                    _TimeoutTimer(IN:=_Step > 0);
IF _TimeoutTimer.Q THEN
	_Step := 0;
	_Error := TRUE;
	_ErrorDescription := 'timed out waiting for response.';
END_IF

_ResetRtrig(CLK:=_Reset);
IF _ResetRtrig.Q THEN
	_Reset := FALSE;
	_Step := 0;
END_IF

_Done := _Step = 0;
_Busy := NOT _Done;

CASE _Step OF
	0: // IDLE
		IF _Execute AND NOT _PythonTcpClient.bBusyWrite THEN
			_Execute := FALSE;
			_Step := _Step + 1;
		ELSIF _Execute THEN
			_Execute := FALSE;
		END_IF
	
	1: // CALL
		_ReadRecordLast := _PythonTcpClient.bRecordRead;
		IF _PythonTcpClient.M_Write(Data:=_Command) THEN
			_Step := _Step + 1;
		ELSE
			_Error := TRUE;
			_ErrorDescription := 'tcp client busy or not connected';
			_Step := 0;
		END_IF
	
	2: // WAIT
		IF _PythonTcpClient.bRecordRead <> _ReadRecordLast THEN
			_ReadRecordLast := _PythonTcpClient.bRecordRead;
			IF find(_PythonTcpClient.strRead, 'res: ') = 1 THEN
				MemUtils.MemSet(
					pbyBuffer:=ADR(_Response),
					byValue:=0,
					dwSize:=SIZEOF(_Response));
				_Response := _PythonTcpClient.strRead;
				_Step := 0;
				
			ELSIF find(_PythonTcpClient.strRead, 'worker uid: ') = 1 THEN
				MemUtils.MemSet(
					pbyBuffer:=ADR(_WorkerUid),
					byValue:=0,
					dwSize:=SIZEOF(_WorkerUid));
				_WorkerUid := DELETE(STR:=_PythonTcpClient.strRead, LEN:=12, POS:=1);
				
			ELSIF find(_PythonTcpClient.strRead, 'command uid: ') = 1 THEN
				MemUtils.MemSet(
					pbyBuffer:=ADR(_WorkerUid),
					byValue:=0,
					dwSize:=SIZEOF(_WorkerUid));
				_WorkerUid := DELETE(STR:=_PythonTcpClient.strRead, LEN:=12, POS:=1);
				
			END_IF
		END_IF
		
END_CASE

_PythonTcpClient(
	bEnable:= TRUE, 
	strIpAddress:= sIpAddress, 
	uPort:= uPort,
	bBusyWrite=> , 
	bDoneWrite=> , 
	bBusyRead=> , 
	bRecordRead=> , 
	strRead=> );
                  

METHOD PUBLIC M_Reset : BOOL
VAR_INPUT
END_VAR
                          _Reset := TRUE;
_Error := FALSE;
_ErrorDescription := '';
                        
END_METHOD

METHOD PUBLIC M_CalibrateCamera : BOOL
VAR_INPUT
	iImageWidth: UINT:=2016;
	iImageHeight: UINT:=2000;
	uTimeout: UDINT:=60; //sec
	fCalCheckerSize: REAL:=25.0; //mm
	iCalCheckerX: UINT:=6;
	iCalCheckerY: UINT:=9;
END_VAR
VAR	
	_CalScriptFileName: STRING:='/var/opt/codesys/PlcLogic/Application/Vision/CalibrateCamera.py';
	_CalResultFile: STRING:='/var/opt/codesys/PlcLogic/visu/outputimage.jpg';
END_VAR
                          
// calibrate with a checkerboard
// sudo python /var/opt/codesys/PlcLogic/Application/CalibrateCamera.py -s cal.yaml -l 24.5 -x 6 -y 9 -d false

IF NOT _Busy THEN
	M_CalibrateCamera := TRUE;
	
	_TimeoutTimer.PT := UDINT_TO_TIME(uTimeout * 1000);
	
	_Command := CONCAT('sudo python ', _CalScriptFileName);
	_Command := CONCAT(_Command, ' -l ');
	_Command := CONCAT(_Command, REAL_TO_STRING(fCalCheckerSize));
	_Command := CONCAT(_Command, ' -x ');
	_Command := CONCAT(_Command, UINT_TO_STRING(iCalCheckerX));
	_Command := CONCAT(_Command, ' -y ');
	_Command := CONCAT(_Command, UINT_TO_STRING(iCalCheckerY));
	_Command := CONCAT(_Command, ' -w ');
	_Command := CONCAT(_Command, UINT_TO_STRING(iImageWidth));
	_Command := CONCAT(_Command, ' -h ');
	_Command := CONCAT(_Command, UINT_TO_STRING(iImageHeight));
	_Command := CONCAT(_Command, ' -r ');
	_Command := CONCAT(_Command, _CalResultFile);
	_Command := CONCAT(_Command, ' 2> ./vision_log.txt ');
	_Execute := TRUE;
	
ELSE
	M_CalibrateCamera := FALSE;
	//_Error := TRUE;
	//_ErrorDescription := 'function busy.';
	
END_IF
                        
END_METHOD

METHOD PUBLIC M_Cancel : BOOL
VAR_INPUT
END_VAR
                          IF _WorkerUid <> '' THEN
	M_Cancel := TRUE;
	_Command := 'kill: ';
	_Command := CONCAT(_Command, _WorkerUid);
	_WorkerUid := ''; // lets make sure to forget this uid in case its used again for something else
	_Step := 0;
	_Execute := TRUE;
	
ELSE
	M_Cancel := FALSE;
	
END_IF
                        
END_METHOD

METHOD PUBLIC M_CaptureImage : BOOL
VAR_INPUT
	iImageWidth: UINT:=2016;
	iImageHeight: UINT:=2000;
	uTimeout: UDINT:=60; //sec
END_VAR
VAR
	_ImageScriptFileName: STRING:='/var/opt/codesys/PlcLogic/Application/Vision/CaptureImage.py';
	_CaptureImageName: STRING:='/var/opt/codesys/PlcLogic/visu/outputimage.jpg';
END_VAR
                          
// capture an image
// sudo python /var/opt/codesys/PlcLogic/Application/CaptureImage.py -s /var/opt/codesys/PlcLogic/Application/input.jpg -w 2016 -h 2000

IF NOT _Busy THEN
	M_CaptureImage := TRUE;
	
	_TimeoutTimer.PT := UDINT_TO_TIME(uTimeout * 1000);
	
	_Command := CONCAT('sudo python ', _ImageScriptFileName);
	_Command := CONCAT(_Command, ' -s ');
	_Command := CONCAT(_Command, _CaptureImageName);
	_Command := CONCAT(_Command, ' -w ');
	_Command := CONCAT(_Command, UINT_TO_STRING(iImageWidth));
	_Command := CONCAT(_Command, ' -h ');
	_Command := CONCAT(_Command, UINT_TO_STRING(iImageHeight));
	_Command := CONCAT(_Command, ' 2> ./vision_log.txt '); 
	_Execute := TRUE;
	
ELSE
	M_CaptureImage := FALSE;
	//_Error := TRUE;
	//_ErrorDescription := 'function busy.';
	
END_IF

                        
END_METHOD

METHOD PUBLIC M_LocatePart : BOOL
VAR_INPUT
	iImageWidth: UINT:=2016;
	iImageHeight: UINT:=2000;
	uTimeout: UDINT:=60; //sec
	iMaxPos: UINT:=10; // i
	dMaxOverlap: REAL:=0.0; // j
	dScore: REAL:=0.8; // k
	dToleranceAngle: REAL:=90.0; // l
	sTemplateName: STRING:='template.jpg';
	sScriptFilename: STRING:='FastTemplateMatching.py';
END_VAR
VAR CONSTANT
	//_SCRIPT_FILE_NAME: STRING:='/var/opt/codesys/PlcLogic/Application/Vision/FastTemplateMatching.py';
	_SCRIPT_DIR_PATH: STRING:='/var/opt/codesys/PlcLogic/Application/Vision/';
	_RESULT_FILE_NAME: STRING:='/var/opt/codesys/PlcLogic/visu/outputimage.jpg';
	_TEMPLATE_DIR_PATH: STRING:='/var/opt/codesys/PlcLogic/Application/Vision/Templates/';
END_VAR
                          
// run the designated vision program
// sudo python /var/opt/codesys/PlcLogic/Application/Vision/TemplateMatch.py -s /var/opt/codesys/PlcLogic/visu/outputimage.jpg        -t /var/opt/codesys/PlcLogic/Application/Vision/Template3.JPG -i 0.9 -j 1.0 -d true -w 2016 -h 2000
// sudo python /var/opt/codesys/PlcLogic/Application/Vision/FastTemplateMatching.py -s /var/opt/codesys/PlcLogic/visu/outputimage.jpg -t /var/opt/codesys/PlcLogic/Application/Vision/Template.jpg -w 2016 -h 2000 -d false
IF NOT _Busy THEN
	M_LocatePart := TRUE;
	
	_TimeoutTimer.PT := UDINT_TO_TIME(uTimeout * 1000);
	
	_Command := CONCAT('sudo python ', _SCRIPT_DIR_PATH);
	_Command := CONCAT(_Command, sScriptFilename);
	//_Command := CONCAT(_Command, ' -s '); // need to trim down the string length
	//_Command := CONCAT(_Command, _VisionImageName);
	_Command := CONCAT(_Command, ' -t ');
	_Command := CONCAT(_Command, _TEMPLATE_DIR_PATH);
	_Command := CONCAT(_Command, sTemplateName);
	_Command := CONCAT(_Command, ' -i ');
	_Command := CONCAT(_Command, UINT_TO_STRING(iMaxPos));
	_Command := CONCAT(_Command, ' -j ');
	_Command := CONCAT(_Command, REAL_TO_STRING(dMaxOverlap));
	_Command := CONCAT(_Command, ' -k ');
	_Command := CONCAT(_Command, REAL_TO_STRING(dScore));
	_Command := CONCAT(_Command, ' -l ');
	_Command := CONCAT(_Command, REAL_TO_STRING(dToleranceAngle));
	_Command := CONCAT(_Command, ' -w ');
	_Command := CONCAT(_Command, UINT_TO_STRING(iImageWidth));
	_Command := CONCAT(_Command, ' -h ');
	_Command := CONCAT(_Command, UINT_TO_STRING(iImageHeight));
	_Command := CONCAT(_Command, ' 2> ./vision_log.txt ');
	_Execute := TRUE;
	
ELSE
	M_LocatePart := FALSE;
	//_Error := TRUE;
	//_ErrorDescription := 'function busy.';
	
END_IF
                        
END_METHOD

{attribute 'monitoring':='variable'}
PROPERTY PUBLIC P_Busy : BOOL
GET
VAR
END_VAR
                            P_Busy := _Busy;
                          
END_GET
END_PROPERTY

{attribute 'monitoring':='variable'}
PROPERTY PUBLIC P_Done : BOOL
GET
VAR
END_VAR
                            P_Done := _Done;
                          
END_GET
END_PROPERTY

{attribute 'monitoring':='variable'}
PROPERTY PUBLIC P_Result : STRING(255)
GET
VAR
END_VAR
                            P_Result := _Response;
                          
END_GET
END_PROPERTY

PROPERTY PUBLIC P_Error : BOOL
GET
VAR
END_VAR
                            P_Error := _Error;
                          
END_GET
END_PROPERTY

PROPERTY PUBLIC P_ErrorDescription : STRING
GET
VAR
END_VAR
                            P_ErrorDescription := _ErrorDescription;
                          
END_GET
END_PROPERTY
END_FUNCTION_BLOCK

FUNCTION_BLOCK PythonTcpClient
VAR_INPUT
	bEnable: BOOL;
	strIpAddress: STRING(19):='127.0.0.1';
	uPort: UINT:=50011;
END_VAR
VAR
	_Write: BOOL:=FALSE;
	_DataToWrite: STRING(255):='';
END_VAR
VAR_OUTPUT
	bBusyWrite: BOOL;
	bDoneWrite: BOOL;
	bBusyRead: BOOL;
	bRecordRead: DINT;
	strRead: STRING(255);
	bConnected: BOOL;
END_VAR

VAR
    _ipAddress       : NBS.IPv4Address;
    _fbTcpClient     : NBS.TCP_Client;
    _fbTcpRead       : NBS.TCP_Read;
    _fbTcpWrite      : NBS.TCP_Write;	
	
	_ConnectDelayTimer: TON;
	_WriteRetriesMax: INT:=3;
	_WriteRetriesCount: INT;
	_WriteRetry: BOOL;
	
	_WriteData: StringByteArray;
	_ReadData: StringByteArray;
	//_TxString: STRING(255);
	//_RxString: STRING(255);
	
	_WriteRTRIG: R_TRIG;
	_ConnectStep, _WriteStep, _ReadStep: INT;
	_Read: BOOL;
END_VAR

VAR CONSTANT
	ConnectStep_IDLE: 	INT:=00;
	ConnectStep_DELAY: 	INT:=10;
	ConnectStep_SETUP: 	INT:=20;
	ConnectStep_ENABLE: INT:=30;
	ConnectStep_WAIT: 	INT:=40;
	ConnectStep_CONN: 	INT:=50;
END_VAR

VAR CONSTANT
	WriteStep_IDLE: 	INT:=00;
	WriteStep_DATA: 	INT:=10;
	WriteStep_WRITE: 	INT:=20;
	WriteStep_WAIT: 	INT:=30;
END_VAR

VAR CONSTANT
	ReadStep_RESET: 	INT:=00;
	ReadStep_IDLE: 		INT:=10;
	ReadStep_ENABLE: 	INT:=20;
	ReadStep_MONITOR: 	INT:=30;
END_VAR

                    {region "connect"}
	
	bConnected := (_ConnectStep = ConnectStep_CONN);
	_ConnectDelayTimer(IN:=_ConnectStep = ConnectStep_DELAY, PT:=T#1S);
	CASE _ConnectStep OF
		
		ConnectStep_IDLE: // IDLE
			IF bEnable THEN
				_fbTcpClient.xEnable := FALSE;
				_ConnectStep := ConnectStep_DELAY;
			END_IF
			
		ConnectStep_DELAY: // DELAY
			IF _ConnectDelayTimer.Q THEN
				_ConnectStep := ConnectStep_SETUP;
			END_IF
			
		ConnectStep_SETUP: // SETUP
			_ipAddress.SetInitialValue(ipAddress := strIpAddress);
			_ConnectStep := ConnectStep_ENABLE;
			
		ConnectStep_ENABLE: // ENABLE
			_fbTcpClient.xEnable := TRUE;
			_ConnectStep := ConnectStep_WAIT;
			
		ConnectStep_WAIT: // WAIT
			IF _fbTcpClient.xActive THEN
				_ConnectStep := ConnectStep_CONN;
			ELSIF _fbTcpClient.xError THEN
				_ConnectStep := ConnectStep_IDLE;
			END_IF
		
		ConnectStep_CONN: // CONNECTED
			IF _fbTcpClient.xError OR NOT _fbTcpClient.xActive OR NOT bEnable THEN
				_ConnectStep := ConnectStep_IDLE;
			END_IF
			
	END_CASE
	
	_fbTcpClient(
		xEnable := , 
		itfIPAddress := _ipAddress, 
		uiPort := uPort, 
		udiTimeOut := 1000000); // us
			 
{endregion}


{region "write"}
	_WriteRTRIG(CLK:=_Write);
	CASE _WriteStep OF
			
		WriteStep_IDLE: // IDLE
			IF (_WriteRTRIG.Q OR _WriteRetry) AND bConnected THEN
				_Write := FALSE;
				_WriteRetry := FALSE;
				_fbTcpWrite.xExecute := FALSE;
				_WriteStep := WriteStep_DATA;
			END_IF
			
		WriteStep_DATA: // DATA
			IF _DataToWrite <> '' THEN
				MemUtils.MemSet(
					pbyBuffer:=ADR(_WriteData.bArray),
					byValue:=0,
					dwSize:=SIZEOF(_WriteData.bArray));
				MemUtils.MemCpy(
					pbyDest:=ADR(_WriteData.sString),
					pbySrc:=ADR(_DataToWrite),
					dwSize:=INT_TO_DWORD(LEN(_DataToWrite)));
				_WriteStep := WriteStep_WRITE;
			ELSE
				_WriteStep := WriteStep_IDLE;
			END_IF
			
		WriteStep_WRITE: // WRITE
			_fbTcpWrite.xExecute := TRUE;
			_WriteStep := WriteStep_WAIT;
		
		WriteStep_WAIT: // WAIT
			IF _fbTcpWrite.xDone THEN
				_fbTcpWrite.xExecute := FALSE;
				_WriteRetriesCount := 0;
				_WriteStep := WriteStep_IDLE;
				
			ELSIF _fbTcpWrite.xError THEN
				IF _WriteRetriesCount <= _WriteRetriesMax THEN
					_WriteRetriesCount := _WriteRetriesCount + 1;
					_WriteRetry := TRUE;
					_WriteStep := WriteStep_IDLE;
					
				ELSIF _WriteRetriesCount > _WriteRetriesMax THEN
					_WriteRetriesCount := 0;
					_WriteStep := WriteStep_IDLE;
					
				END_IF
			END_IF
	END_CASE
	
	bBusyWrite := ((_WriteStep <> WriteStep_IDLE) OR _WriteRetry) AND _fbTcpWrite.xBusy;
	bDoneWrite := (_WriteStep = WriteStep_IDLE) AND _fbTcpWrite.xDone;
	_fbTcpWrite(xExecute := ,
				itfConnection := _fbTcpClient.itfConnection, 
				udiTimeOut := 1000000, // us 
				udiSize := INT_TO_UDINT(LEN(_WriteData.sString)), 
				pData := ADR(_WriteData.bArray));

{endregion}


{region "read"}

	_Read := (_ConnectStep = ConnectStep_CONN);
	CASE _ReadStep OF
			 
		ReadStep_RESET: // RESET
			_fbTcpRead.xEnable := FALSE;
			_ReadStep := ReadStep_IDLE;

		ReadStep_IDLE: // IDLE
			IF _Read THEN
				_ReadStep := ReadStep_ENABLE;
			END_IF

		ReadStep_ENABLE: // ENABLE
			_fbTcpRead.xEnable := TRUE;
			_ReadStep := ReadStep_MONITOR;

		ReadStep_MONITOR: // MONITOR
			IF _fbTcpRead.xReady THEN
				IF (_fbTcpRead.udiCount > 0) THEN
					//
					MemUtils.MemSet(
						pbyBuffer:=ADR(strRead),
						byValue:=0,
						dwSize:=SIZEOF(strRead)); 
					MemUtils.MemCpy(
						pbyDest:=ADR(strRead),
						pbySrc:=ADR(_ReadData.sString),
						dwSize:=SEL(_fbTcpRead.udiCount > 255, _fbTcpRead.udiCount, 255));
					MemUtils.MemSet(
						pbyBuffer:=ADR(_ReadData.sString),
						byValue:=0,
						dwSize:=SIZEOF(_ReadData.sString)); 
					//
					bRecordRead := bRecordRead + 1;
				END_IF
				
			ELSIF _fbTcpRead.xError OR NOT _Read THEN
				_ReadStep := ReadStep_RESET;
				
			END_IF
			 
	END_CASE
	
	bBusyRead := (_ReadStep <> ReadStep_IDLE) AND _fbTcpRead.xBusy;
	_fbTcpRead(xEnable := , 
				itfConnection := _fbTcpClient.itfConnection, 
				udiSize := SIZEOF(_ReadData.bArray), 
				pData := ADR(_ReadData.bArray), 
				udiCount => );

{endregion}
                  

METHOD PUBLIC M_Write : BOOL
VAR_INPUT
	Data: STRING(255);
END_VAR
                          IF bConnected AND NOT bBusyWrite THEN
	_Write:=TRUE;
	_DataToWrite:=Data;
	M_Write := TRUE;
	
ELSE
	M_Write := FALSE;
	
END_IF
                        
END_METHOD
END_FUNCTION_BLOCK

FUNCTION_BLOCK ParseVisionCmd
VAR_INPUT
    Command: STRING(GVL.COMMAND_LEN);
END_VAR
VAR_OUTPUT
    stCommand: ST_VisionCmd;
	Error: BOOL;
	ErrorDescription: STRING;
END_VAR
VAR
	_CmdParams: ARRAY [0..GVL.COMMAND_LEN] OF STRING;
    _CommandType: STRING;
	_StrPosition: INT;
END_VAR
VAR CONSTANT
	_CommandTypeCal: STRING(3):='CAL'; // calibrate vision
	_CommandTypeAcq: STRING(3):='ACQ'; // acquire (capture) image
	_CommandTypeLoc: STRING(3):='LOC'; // locate part
END_VAR

                    // C|A|L ImageWidth ImageHeight Timeout

// C Calibrate vision system
    // CheckerSize (user units) XCount YCount 
    // C 2016 2000 60 25.0 6 9
    
// A Aquire image
    // A 2016 2000 60
    
// L Locate part 
    // MaxParts MaxOverlap Score ToleranceAngle ResultPostion TemplateName ScriptName
    // L 2016 2000 60 10 0.0 0.8 90.0 1 template.jpg FastTemplateMatching.py
	// MaxParts - max number of parts to find in image
	// MaxOverlap - max overlap of parts in image
	// Score - min required score for parts
	// ToleranceAngle - +/- search angle (the larger the number, the longer the search)
	// ResultPostion - index of vision register to store result
	// TemplateName - name of the template to search for
	// ScriptName - name of the template to search for

Error:=FALSE;
ErrorDescription:='';

// split command string into commands
_CmdParams:=F_SplitCmd(Command:=Command);

_CommandType:= _CmdParams[0];
IF _CommandType = _CommandTypeCal THEN
    // C 2016 2000 0060 025.0 0006 0009
	stCommand.CommandType:=DUT_Command_VisionType.Calibrate;
    stCommand.Calibrate.CheckerSize:=STRING_TO_REAL(_CmdParams[4]);
    stCommand.Calibrate.CheckerXCount:=STRING_TO_UINT(_CmdParams[5]);
    stCommand.Calibrate.CheckerYCount:=STRING_TO_UINT(_CmdParams[6]);
	
	IF stCommand.Calibrate.CheckerSize <= 0
		OR stCommand.Calibrate.CheckerXCount <= 0
		OR stCommand.Calibrate.CheckerYCount <= 0 THEN
			Error:=TRUE;
			ErrorDescription:='Checkerboard configuration incorrect';
			RETURN;
	END_IF
    
ELSIF _CommandType = _CommandTypeAcq THEN
    // A 2016 2000 0060
	stCommand.CommandType:=DUT_Command_VisionType.Acquire;
    
ELSIF _CommandType = _CommandTypeLoc THEN
    // L 2016 2000 0060 0010 000.0 0.8 090.0 001 template.jpg FastTemplatMatching.py
	stCommand.CommandType:=DUT_Command_VisionType.LocatePart;
    stCommand.Locate.MaxParts:=STRING_TO_UINT(_CmdParams[4]);
    stCommand.Locate.MaxOverlap:=STRING_TO_REAL(_CmdParams[5]);
    stCommand.Locate.Score:=STRING_TO_REAL(_CmdParams[6]);
    stCommand.Locate.ToleranceAngle:=STRING_TO_REAL(_CmdParams[7]);
    stCommand.Locate.ResultPosition:=STRING_TO_UINT(_CmdParams[8]);
    stCommand.Locate.TemplateName:=_CmdParams[9];
    stCommand.Locate.ScriptFilename:=_CmdParams[10];
	
	IF stCommand.Locate.MaxParts <= 0
		OR stCommand.Locate.ResultPosition < GVL.VIS_ARR_BEG
		OR stCommand.Locate.ResultPosition > GVL.VIS_ARR_END
		OR stCommand.Locate.TemplateName = '' THEN
			Error:=TRUE;
			ErrorDescription:='Locate part configuration incorrect';
			RETURN;
	END_IF
	
ELSE
	Error:=TRUE;
	ErrorDescription:='Unknown command type for vision';
	RETURN;
    
END_IF

// common
stCommand.ImageWidth:=STRING_TO_UINT(_CmdParams[1]);
stCommand.ImageHeight:=STRING_TO_UINT(_CmdParams[2]);
stCommand.Timeout:=STRING_TO_UDINT(_CmdParams[3]);

IF stCommand.ImageWidth <= 0
	OR stCommand.ImageHeight <= 0 THEN
		Error:=TRUE;
		ErrorDescription:='Image size settings incorrect';
END_IF
                  
END_FUNCTION_BLOCK

FUNCTION BuildVisionCmd : STRING(GVL.COMMAND_LEN)
VAR_INPUT
    stCommand: ST_VisionCmd;
END_VAR
VAR
    _Command: STRING(GVL.COMMAND_LEN);
END_VAR
VAR CONSTANT
	_Delimiter: STRING:=' ';
	_CommandTypeCal: STRING(3):='CAL'; // calibrate vision
	_CommandTypeAcq: STRING(3):='ACQ'; // acquire (capture) image
	_CommandTypeLoc: STRING(3):='LOC'; // locate part
END_VAR

                    // C|A|L ImageWidth ImageHeight Timeout

// C Calibrate vision system
    // CheckerSize (user units) XCount YCount 
    // C 2016 2000 60 25.0 6 9
    
// A Aquire image
    // A 2016 2000 60
    
// L Locate part 
    // MaxParts MaxOverlap Score ToleranceAngle ResultPostion TemplateName ScriptName
    // L 2016 2000 60 10 0.0 0.8 90.0 1 template.jpg FastTemplateMatching.py
	// MaxParts - max number of parts to find in image
	// MaxOverlap - max overlap of parts in image
	// Score - min required score for parts
	// ToleranceAngle - +/- search angle (the larger the number, the longer the search)
	// ResultPostion - index of vision register to store result
	// TemplateName - name of the template to search for
	// ScriptName - name of the template to search for

// clear the command
_Command:='';

// build the command
CASE stCommand.CommandType OF
	DUT_Command_VisionType.Calibrate:
		F_AddElement(_Command, _Delimiter, _CommandTypeCal);
	DUT_Command_VisionType.Acquire:
		F_AddElement(_Command, _Delimiter, _CommandTypeAcq);
	DUT_Command_VisionType.LocatePart:
		F_AddElement(_Command, _Delimiter, _CommandTypeLoc);
END_CASE

// add the common items width, height, timeout
F_AddElement(_Command, _Delimiter, UINT_TO_STRING(stCommand.ImageWidth));
F_AddElement(_Command, _Delimiter, UINT_TO_STRING(stCommand.ImageHeight));
F_AddElement(_Command, _Delimiter, UDINT_TO_STRING(stCommand.Timeout));

//
CASE stCommand.CommandType OF
	DUT_Command_VisionType.Calibrate:
		// C 2016 2000 60 25.0 6 9
		F_AddElement(_Command, _Delimiter, REAL_TO_STRING(stCommand.Calibrate.CheckerSize));
		F_AddElement(_Command, _Delimiter, UINT_TO_STRING(stCommand.Calibrate.CheckerXCount));
		F_AddElement(_Command, _Delimiter, UINT_TO_STRING(stCommand.Calibrate.CheckerYCount));
		
	DUT_Command_VisionType.Acquire:
		// A 2016 2000 60
		// we are done
		
	DUT_Command_VisionType.LocatePart:
		// L 2016 2000 60 10 0.0 0.8 90.0 1 template.jpg FastTemplateMatching.py
		F_AddElement(_Command, _Delimiter, UINT_TO_STRING(stCommand.Locate.MaxParts));
		F_AddElement(_Command, _Delimiter, REAL_TO_STRING(stCommand.Locate.MaxOverlap));
		F_AddElement(_Command, _Delimiter, REAL_TO_STRING(stCommand.Locate.Score));
		F_AddElement(_Command, _Delimiter, REAL_TO_STRING(stCommand.Locate.ToleranceAngle));
		F_AddElement(_Command, _Delimiter, UINT_TO_STRING(stCommand.Locate.ResultPosition));
		F_AddElement(_Command, _Delimiter, stCommand.Locate.TemplateName);
		F_AddElement(_Command, _Delimiter, stCommand.Locate.ScriptFilename);
		
END_CASE

// set function equal to command
BuildVisionCmd := _Command;
                  
END_FUNCTION

FUNCTION_BLOCK Module EXTENDS PackML IMPLEMENTS ItfModule

VAR_INPUT // input vars
	StoredPositions: REFERENCE TO ARRAY[GVL.POS_ARR_BEG..GVL.POS_ARR_END] OF DUT_StoredPosition;
	VisionRegisters: REFERENCE TO ARRAY[GVL.VIS_ARR_BEG..GVL.VIS_ARR_END] OF DUT_VisionRegister;
	Flags: REFERENCE TO ARRAY[GVL.FLG_ARR_BEG..GVL.FLG_ARR_END] OF DUT_Flags;
END_VAR

VAR_OUTPUT // output vars
	ItfUnitMode: PACK_ML.IUnitMode;
	Busy: BOOL;
	Error: BOOL;
	ErrorDescription: STRING;
END_VAR

VAR // standard local vars
	_TimeoutTimer: TON:=(PT:=T#120S);
	_Home, _Start: BOOL;
	_ModuleFirstScan: BOOL:=TRUE;
	_SeqStart, _SeqHome: INT;
	_AbortedRtrig: R_Trig;
END_VAR

VAR CONSTANT //
	STEP_IDLE: INT := 0000;
	STEP_DONE: INT := 0020;
	STEP_RUN:  INT := 0030;
END_VAR

                    SUPER^();

//
IF _ModuleFirstScan THEN
	ItfUnitMode := SUPER^.IUnitMode;
END_IF;

//
_M_Home();
_M_Start();

//
Busy := _UnitMode.CurrentState <> PACK_ML.State.Idle
		AND _UnitMode.CurrentState <> PACK_ML.State.Aborted
		AND _UnitMode.CurrentState <> PACK_ML.State.Complete
		AND _UnitMode.CurrentState <> PACK_ML.State.Held
		AND _UnitMode.CurrentState <> PACK_ML.State.Stopped
		AND _UnitMode.CurrentState <> PACK_ML.State.Suspended;
		
//
_AbortedRtrig(CLK:=_UnitMode.CurrentState = PACK_ML.State.Aborted);
IF _AbortedRtrig.Q THEN
	//_SeqStart := 0;  _Start:=FALSE;
	//_SeqHome := 0; _Home:=FALSE;
END_IF

//
_TimeoutTimer(IN:= Busy);
IF _TimeoutTimer.Q THEN
	M_Error(Description:= CONCAT('Task timed out after ', TIME_TO_STRING(_TimeoutTimer.ET)));
END_IF

// do not place anything below this
_ModuleFirstScan:=FALSE;
                  

METHOD PUBLIC M_Start
VAR_INPUT
END_VAR
                          _Start := TRUE;
                        
END_METHOD

METHOD PUBLIC M_Home
VAR_INPUT
END_VAR
                          _Home:=TRUE;
                        
END_METHOD

METHOD PROTECTED M_Error : BOOL
VAR_INPUT
	Description: STRING;
END_VAR
                          // suspend state machine
_UnitMode.Suspend();

//
Error := TRUE;

//
IF ErrorDescription = '' THEN
	ErrorDescription := Description;
ELSE // add a space and tack on the additional error description
	ErrorDescription := CONCAT(ErrorDescription, ' ');
	ErrorDescription := CONCAT(ErrorDescription, Description);
END_IF
                        
END_METHOD

METHOD PUBLIC M_Abort
VAR_INPUT
END_VAR
                          _UnitMode.Abort();
_SeqStart := 0;  _Start:=FALSE;
_SeqHome := 0; _Home:=FALSE;
                        
END_METHOD

METHOD PUBLIC M_Hold
VAR_INPUT
END_VAR
                          _UnitMode.Hold();
                        
END_METHOD

METHOD PUBLIC M_Stop
VAR_INPUT
END_VAR
                          _UnitMode.Stop();
                        
END_METHOD

METHOD PRIVATE _M_Start : BOOL
                          CASE _SeqStart OF
	0:
		IF _Start THEN
			_Start := FALSE;
			M_Reset();
			_SeqStart := _SeqStart + 1;
		END_IF
	1:
		CASE _UnitMode.CurrentState OF
			PACK_ML.State.Clearing,
			PACK_ML.State.Resetting,
			PACK_ML.State.UnHolding,
			PACK_ML.State.UnSuspending,
			PACK_ML.State.Starting:
				// be patient
			PACK_ML.State.Aborted:
				_UnitMode.Clear();
			PACK_ML.State.Stopped:
				_UnitMode.Reset();
			PACK_ML.State.Held:
				_UnitMode.UnHold();
			PACK_ML.State.Suspended:
				_UnitMode.UnSuspend();
			PACK_ML.State.Idle:
				_UnitMode.Start();
			PACK_ML.State.Execute:
				_SeqStart := 0;
		ELSE
			_SeqStart := 0;
		END_CASE
		
END_CASE
                        
END_METHOD

METHOD PROTECTED M_Reset : BOOL
VAR_INPUT
END_VAR
                          Error := FALSE;
ErrorDescription := '';
                        
END_METHOD

METHOD PRIVATE _M_Home : BOOL
                          CASE _SeqHome OF
	0:
		//
		IF _Home THEN
			_Home := FALSE;
			M_Reset();
			_SeqHome := _SeqHome + 1;
		END_IF
	1:
		//
		CASE _UnitMode.CurrentState OF
			PACK_ML.State.Aborted:
				_UnitMode.Clear();
				
			PACK_ML.State.Stopped,
			PACK_ML.State.Complete:
				_UnitMode.Reset();
				_SeqHome := _SeqHome + 1;
				
			PACK_ML.State.Resetting,
			PACK_ML.State.Clearing,
			PACK_ML.State.Aborting:
				// just wait
		ELSE
			_UnitMode.Abort();
			
		END_CASE
		
	2:
		IF _UnitMode.CurrentState = PACK_ML.State.Idle THEN
			_SeqHome := 0;
		END_IF
		
END_CASE
                        
END_METHOD

{attribute 'monitoring' := 'variable'}
PROPERTY PropCurrentState : PACK_ML.State
GET
VAR
END_VAR
                            PropCurrentState := ItfUnitMode.CurrentState;
                          
END_GET
END_PROPERTY

{attribute 'monitoring' := 'variable'}
PROPERTY PropBusy : BOOL
GET
VAR
END_VAR
                            PropBusy := Busy;
                          
END_GET
END_PROPERTY

{attribute 'monitoring' := 'variable'}
PROPERTY PropError : BOOL
GET
VAR
END_VAR
                            PropError := Error;
                          
END_GET
END_PROPERTY

{attribute 'monitoring' := 'variable'}
PROPERTY PropErrDescription : STRING
GET
VAR
END_VAR
                            PropErrDescription := ErrorDescription;
                          
END_GET
END_PROPERTY
END_FUNCTION_BLOCK

FUNCTION_BLOCK VisionCmdProcessor EXTENDS Module
VAR_INPUT
	Command: STRING(GVL.COMMAND_LEN):='';
END_VAR
VAR_OUTPUT
	VisionStateText: STRING:='READY';
END_VAR
VAR
	_CaptureImage_Output: STRING(255);
	_CaptureImage_WorkerUid: STRING;
	_LocatePart_Output: STRING(255);
	_LocatePart_WorkerUid: STRING;
	_RunCalibration_Output: STRING(255);
	_RunCalibration_WorkerUid: STRING;
    _Vision: OpenCV;
    _VisionCommandParser: ParseVisionCmd;
    _VisionDoneRtrig: R_TRIG;
	_VisionBusyRtrig: R_TRIG;
	_VisionResult: STRING(255);
	_ResultPosition: INT;
	_ResultPosition_CAL: INT;
	_ResultPosition_LOC: INT;
	_ResultPosition_CAP: INT;
	_SpacePosition: INT;
	_VisionObjectIndex: UINT;
	_VisionRatio: REAL;
	_VisionRotation: REAL;
	_VisionError: REAL;
	_UnitModeCurrentState: PACK_ML.State;
END_VAR

VAR CONSTANT
	_RESPONSE_CAL:          STRING:='res: CAL ';
	_RESPONSE_LOC:          STRING:='res: LOC ';
	_RESPONSE_CAP:          STRING:='res: CAP ';

	_STEP_DONE: 			INT := 1000;
	_STEP_IDLE: 			INT := 0000;
	_STEP_COMMAND: 			INT := 0020;
	_STEP_TRIGGER: 			INT := 0030;
	_STEP_WAIT: 			INT := 0040;
	_STEP_ERR: 				INT := 0050;
END_VAR

                    SUPER^();

// PackML state machine implementation
_UnitModeCurrentState := SUPER^._UnitMode.CurrentState;

//
CASE SUPER^._SeqMain OF
	
    _STEP_DONE:
		SUPER^._SeqMain := _STEP_IDLE;
        
    _STEP_IDLE:
		// hang out here until called to run
        
    _STEP_COMMAND: // parse vision command
        _VisionCommandParser(Command:=Command);
		IF _VisionCommandParser.Error THEN
			SUPER^.M_Error(Description:=_VisionCommandParser.ErrorDescription);
			//
			SUPER^._SeqMain := _STEP_ERR;
		ELSE
			IF _VisionCommandParser.stCommand.Timeout > 0 THEN
				SUPER^._TimeoutTimer.PT := UDINT_TO_TIME(_VisionCommandParser.stCommand.Timeout * 1000);
			END_IF
			//
			SUPER^._SeqMain := _STEP_TRIGGER;
		END_IF
		
	_STEP_TRIGGER: //
		CASE _VisionCommandParser.stCommand.CommandType OF
			DUT_Command_VisionType.Calibrate: //
				_Vision.M_CalibrateCamera(	iImageWidth:= _VisionCommandParser.stCommand.ImageWidth, 
											iImageHeight:= _VisionCommandParser.stCommand.ImageHeight, 
											fCalCheckerSize:= _VisionCommandParser.stCommand.Calibrate.CheckerSize, 
											iCalCheckerX:= _VisionCommandParser.stCommand.Calibrate.CheckerXCount, 
											iCalCheckerY:= _VisionCommandParser.stCommand.Calibrate.CheckerYCount,
                                            uTimeout:=_VisionCommandParser.stCommand.Timeout);
			
			DUT_Command_VisionType.Acquire: //
				_Vision.M_CaptureImage(	iImageWidth:= _VisionCommandParser.stCommand.ImageWidth, 
										iImageHeight:= _VisionCommandParser.stCommand.ImageHeight,
                                        uTimeout:=_VisionCommandParser.stCommand.Timeout);
			
			DUT_Command_VisionType.LocatePart: //
				_Vision.M_LocatePart( 	iImageWidth:= _VisionCommandParser.stCommand.ImageWidth, 
										iImageHeight:= _VisionCommandParser.stCommand.ImageHeight, 
										iMaxPos:= _VisionCommandParser.stCommand.Locate.MaxParts, 
										dMaxOverlap:= _VisionCommandParser.stCommand.Locate.MaxOverlap, 
										dScore:= _VisionCommandParser.stCommand.Locate.Score, 
										dToleranceAngle:= _VisionCommandParser.stCommand.Locate.ToleranceAngle,
                                        uTimeout:=_VisionCommandParser.stCommand.Timeout,
										sTemplateName:=_VisionCommandParser.stCommand.Locate.TemplateName,
										sScriptFilename:=_VisionCommandParser.stCommand.Locate.ScriptFilename);
			
		END_CASE;
		
		//
		SUPER^._SeqMain := _STEP_WAIT;
		
	_STEP_WAIT: //
		IF _VisionDoneRtrig.Q THEN
			
			//
			_VisionResult := _Vision.P_Result;
			
			//
			_ResultPosition_CAL := FIND(STR1:=_VisionResult,STR2:=_RESPONSE_CAL);
			_ResultPosition_LOC := FIND(STR1:=_VisionResult,STR2:=_RESPONSE_LOC);
			_ResultPosition_CAP := FIND(STR1:=_VisionResult,STR2:=_RESPONSE_CAP);
			
			//
			IF _ResultPosition_CAL > 0 THEN 
				// calibration was completed
				// res: CAL rat:23.23 rot:23.23 err:23.23
				_VisionResult := MID(STR:=_VisionResult,LEN:=LEN(_VisionResult)-LEN(_RESPONSE_CAL),POS:=LEN(_RESPONSE_CAL)+1);
				//VisionStateText := CONCAT(VisionStateText, '\n');
				//VisionStateText := CONCAT(VisionStateText, _VisionResult);
				// rat:23.23 rot:23.23 err:23.23
				_ResultPosition := FIND(STR1:=_VisionResult,STR2:='rat:');
				IF _ResultPosition > 0 THEN
					_VisionResult := MID(STR:=_VisionResult,LEN:=LEN(_VisionResult)-LEN('rat:'),POS:=LEN('rat:')+1);
					_SpacePosition := FIND(STR1:=_VisionResult,STR2:=' ');
					_VisionRatio := STRING_TO_REAL(MID(STR:=_VisionResult,LEN:=_SpacePosition-1,POS:=1));
					_VisionResult := MID(STR:=_VisionResult,LEN:=LEN(_VisionResult)-_SpacePosition,POS:=_SpacePosition+1);
				END_IF
				// rot:23.23 err:23.23
				_ResultPosition := FIND(STR1:=_VisionResult,STR2:='rot:');
				IF _ResultPosition > 0 THEN
					_VisionResult := MID(STR:=_VisionResult,LEN:=LEN(_VisionResult)-LEN('rot:'),POS:=LEN('rot:')+1);
					_SpacePosition := FIND(STR1:=_VisionResult,STR2:=' ');
					_VisionRotation := STRING_TO_REAL(MID(STR:=_VisionResult,LEN:=_SpacePosition-1,POS:=1));
					_VisionResult := MID(STR:=_VisionResult,LEN:=LEN(_VisionResult)-_SpacePosition,POS:=_SpacePosition+1);
				END_IF
				// err:23.23
				_ResultPosition := FIND(STR1:=_VisionResult,STR2:='err:');
				IF _ResultPosition > 0 THEN
					_VisionResult := MID(STR:=_VisionResult,LEN:=LEN(_VisionResult)-LEN('err:'),POS:=LEN('err:')+1);
					_SpacePosition := FIND(STR1:=_VisionResult,STR2:=' ');
					_VisionError := STRING_TO_REAL(MID(STR:=_VisionResult,LEN:=_SpacePosition-1,POS:=1));
					_VisionResult := MID(STR:=_VisionResult,LEN:=LEN(_VisionResult)-_SpacePosition,POS:=_SpacePosition+1);
				END_IF
				
			ELSIF _ResultPosition_LOC > 0 THEN 
				// part was located
				// 'res: LOC obj:0 cx:54.66 cy:119.45 a:-12.87 s:0.84 $NLOC obj:1 cx:71.49 cy:100.06 a:10.13 s:0.83 $N'
				_VisionResult := MID(STR:=_VisionResult,LEN:=LEN(_VisionResult)-LEN(_RESPONSE_LOC),POS:=LEN(_RESPONSE_LOC)+1);
				//VisionStateText := CONCAT(VisionStateText, '\n');
				//VisionStateText := CONCAT(VisionStateText, _VisionResult);
				_VisionObjectIndex := 0;
				WHILE FIND(STR1:=_VisionResult,STR2:='obj:') > 0 
					AND _VisionObjectIndex <= _VisionCommandParser.stCommand.Locate.MaxParts 
					AND _VisionObjectIndex + _VisionCommandParser.stCommand.Locate.ResultPosition < GVL.VIS_ARR_END DO
					// 'obj:0 cx:54.66 cy:119.45 a:-12.87 s:0.84 $NLOC obj:1 cx:71.49 cy:100.06 a:10.13 s:0.83 $N'
					// $NLOC obj:1 cx:71.49 cy:100.06 a:10.13 s:0.83 $N'
					_ResultPosition := FIND(STR1:=_VisionResult,STR2:='obj:');
					IF _ResultPosition > 0 THEN
						_VisionResult := MID(STR:=_VisionResult,LEN:=LEN(_VisionResult)-_ResultPosition-LEN('obj:')+1,POS:=_ResultPosition+LEN('obj:'));
						_SpacePosition := FIND(STR1:=_VisionResult,STR2:=' ');
						_VisionObjectIndex := STRING_TO_UINT(MID(STR:=_VisionResult,LEN:=_SpacePosition-1,POS:=1));
						SUPER^.VisionRegisters[_VisionCommandParser.stCommand.Locate.ResultPosition + _VisionObjectIndex].Comment := CONCAT('obj:', UDINT_TO_STRING(_VisionObjectIndex));
						_VisionResult := MID(STR:=_VisionResult,LEN:=LEN(_VisionResult)-_SpacePosition,POS:=_SpacePosition+1);
					END_IF
					// cx:54.66 cy:119.45 a:-12.87 s:0.84 $NLOC obj:1 cx:71.49 cy:100.06 a:10.13 s:0.83 $N'
					_ResultPosition := FIND(STR1:=_VisionResult,STR2:='cx:');
					IF _ResultPosition > 0 THEN
						_VisionResult := MID(STR:=_VisionResult,LEN:=LEN(_VisionResult)-LEN('cx:'),POS:=LEN('cx:')+1);
						_SpacePosition := FIND(STR1:=_VisionResult,STR2:=' ');
						SUPER^.VisionRegisters[_VisionCommandParser.stCommand.Locate.ResultPosition + _VisionObjectIndex].Position.X := STRING_TO_LREAL(MID(STR:=_VisionResult,LEN:=_SpacePosition-1,POS:=1));
						_VisionResult := MID(STR:=_VisionResult,LEN:=LEN(_VisionResult)-_SpacePosition,POS:=_SpacePosition+1);
					END_IF
					// cy:119.45 a:-12.87 s:0.84 $NLOC obj:1 cx:71.49 cy:100.06 a:10.13 s:0.83 $N'
					_ResultPosition := FIND(STR1:=_VisionResult,STR2:='cy:');
					IF _ResultPosition > 0 THEN
						_VisionResult := MID(STR:=_VisionResult,LEN:=LEN(_VisionResult)-LEN('cy:'),POS:=LEN('cy:')+1);
						_SpacePosition := FIND(STR1:=_VisionResult,STR2:=' ');
						SUPER^.VisionRegisters[_VisionCommandParser.stCommand.Locate.ResultPosition + _VisionObjectIndex].Position.Y := STRING_TO_LREAL(MID(STR:=_VisionResult,LEN:=_SpacePosition-1,POS:=1));
						_VisionResult := MID(STR:=_VisionResult,LEN:=LEN(_VisionResult)-_SpacePosition,POS:=_SpacePosition+1);
					END_IF
					// a:-12.87 s:0.84 $NLOC obj:1 cx:71.49 cy:100.06 a:10.13 s:0.83 $N'
					_ResultPosition := FIND(STR1:=_VisionResult,STR2:='a:');
					IF _ResultPosition > 0 THEN
						_VisionResult := MID(STR:=_VisionResult,LEN:=LEN(_VisionResult)-LEN('a:'),POS:=LEN('a:')+1);
						_SpacePosition := FIND(STR1:=_VisionResult,STR2:=' ');
						SUPER^.VisionRegisters[_VisionCommandParser.stCommand.Locate.ResultPosition + _VisionObjectIndex].Position.A := STRING_TO_LREAL(MID(STR:=_VisionResult,LEN:=_SpacePosition-1,POS:=1));
						_VisionResult := MID(STR:=_VisionResult,LEN:=LEN(_VisionResult)-_SpacePosition,POS:=_SpacePosition+1);
					END_IF
					// s:0.84 $NLOC obj:1 cx:71.49 cy:100.06 a:10.13 s:0.83 $N'
					_ResultPosition := FIND(STR1:=_VisionResult,STR2:='s:');
					IF _ResultPosition > 0 THEN
						_VisionResult := MID(STR:=_VisionResult,LEN:=LEN(_VisionResult)-LEN('s:'),POS:=LEN('s:')+1);
						_SpacePosition := FIND(STR1:=_VisionResult,STR2:=' ');
						SUPER^.VisionRegisters[_VisionCommandParser.stCommand.Locate.ResultPosition + _VisionObjectIndex].Scaling := STRING_TO_REAL(MID(STR:=_VisionResult,LEN:=_SpacePosition-1,POS:=1));
						_VisionResult := MID(STR:=_VisionResult,LEN:=LEN(_VisionResult)-_SpacePosition,POS:=_SpacePosition+1);
					END_IF
					// $NLOC obj:1 cx:71.49 cy:100.06 a:10.13 s:0.83 $N'
				END_WHILE
				
				
			ELSIF _ResultPosition_CAP > 0 THEN 
				// image was captured
				
			END_IF
			
			//
			SUPER^._SeqMain := _STEP_DONE;
			
		END_IF

END_CASE

//
_Vision(sIpAddress:= '127.0.0.1', uPort:= 50011);

//
_VisionBusyRtrig(clk:=_Vision.P_Busy);
IF _VisionBusyRtrig.Q THEN
	VisionStateText := 'BUSY';
END_IF

//
_VisionDoneRtrig(clk:=_Vision.P_Done);
IF _VisionDoneRtrig.Q THEN
	VisionStateText := 'DONE';
END_IF
                  

METHOD PROTECTED M_SetPackML : BOOL
                          SUPER^._UnitMode(	sName := 'Vision Processor',
				eInitialState := PACK_ML.State.Idle,
				xActive := TRUE);
                        
END_METHOD

METHOD PROTECTED M_Complete : BOOL
                          // once complete, reset to get back to idle
SUPER^._UnitMode.Reset();
                        
END_METHOD

METHOD PROTECTED M_Resetting : BOOL
                          CASE SUPER^._SeqResetting OF
	0:
		_Vision.M_Reset();
		_SeqResetting := _SeqResetting + 1;
	1:
		IF NOT _Vision.P_Error THEN
			VisionStateText := 'RESET';
			SUPER^.M_StateComplete();
			_SeqResetting := 0;
		END_IF
END_CASE
		

                        
END_METHOD

METHOD PROTECTED M_Starting : BOOL
                          // here we want to clear things and get ready for the execute state
// I can consider this the "INIT" state
SUPER^._SeqMain := _STEP_COMMAND;
SUPER^.M_StateComplete();
                        
END_METHOD

METHOD PROTECTED M_Execute : BOOL
                          // here we want to execute our commands/jobs/etc and set completed when done.
IF SUPER^._SeqMain =_STEP_IDLE THEN
	SUPER^.M_StateComplete();
END_IF
                        
END_METHOD

METHOD PROTECTED M_Aborting : BOOL
                          CASE _SeqAborting OF
	0:
		_Vision.M_Cancel();
		_SeqAborting := _SeqAborting + 1;
		
	1: 
		IF NOT _Vision.P_Busy THEN
			SUPER^.M_StateComplete();
			_SeqAborting := 0;
		END_IF
END_CASE
                        
END_METHOD
END_FUNCTION_BLOCK

FUNCTION_BLOCK ParseVarSetCmd
VAR_INPUT
	Command: STRING(GVL.COMMAND_LEN);
END_VAR
VAR_OUTPUT
	stCommand: ST_VarSetCmd;
	Error: BOOL;
	ErrorDescription: STRING;
END_VAR
VAR
	_CmdParams: ARRAY [0..GVL.COMMAND_LEN] OF STRING;
END_VAR
VAR CONSTANT
	_ArrayTypeS: STRING(3):='STO';
	_ArrayTypeV: STRING(3):='VIS';
	_ArrayTypeF: STRING(3):='FLG';
END_VAR

                    // S|V|F index x y z a b c
// S 0000 +0000.00 +0000.00 +0000.00 +0000.00 +0000.00 +0000.00 
// V 0000 +0000.00 +0000.00 +0000.00 +0000.00 +0000.00 +0000.00 
// F 0000 1

Error:=FALSE;
ErrorDescription:='';

// split command string into commands
_CmdParams:=F_SplitCmd(Command:=Command);

//
IF _CmdParams[0] = _ArrayTypeS  THEN
	stCommand.ArrayType := DUT_Command_ArrayType.StoredPosition;
ELSIF _CmdParams[0] = _ArrayTypeV THEN
	stCommand.ArrayType := DUT_Command_ArrayType.VisionRegister;
ELSIF _CmdParams[0] = _ArrayTypeF THEN
	stCommand.ArrayType := DUT_Command_ArrayType.Flag;
ELSE
	Error:=TRUE;
	ErrorDescription:='Incorrect array type';
END_IF

//
stCommand.ArrayIndex := STRING_TO_INT(_CmdParams[1]);
IF ((stCommand.ArrayIndex < GVL.POS_ARR_BEG OR stCommand.ArrayIndex > GVL.POS_ARR_END) AND stCommand.ArrayType = DUT_Command_ArrayType.StoredPosition)
	OR ((stCommand.ArrayIndex < GVL.VIS_ARR_BEG OR stCommand.ArrayIndex > GVL.VIS_ARR_END) AND stCommand.ArrayType = DUT_Command_ArrayType.VisionRegister)
	OR ((stCommand.ArrayIndex < GVL.FLG_ARR_BEG OR stCommand.ArrayIndex > GVL.FLG_ARR_END) AND stCommand.ArrayType = DUT_Command_ArrayType.Flag) THEN
		Error:=TRUE;
		ErrorDescription:='Incorrect array type';
END_IF

//
stCommand.Coordinates.X := STRING_TO_LREAL(_CmdParams[2]);
stCommand.Coordinates.Y := STRING_TO_LREAL(_CmdParams[3]);
stCommand.Coordinates.Z := STRING_TO_LREAL(_CmdParams[4]);
stCommand.Coordinates.A := STRING_TO_LREAL(_CmdParams[5]);
stCommand.Coordinates.B := STRING_TO_LREAL(_CmdParams[6]);
stCommand.Coordinates.C := STRING_TO_LREAL(_CmdParams[7]);
                  
END_FUNCTION_BLOCK

FUNCTION_BLOCK MoveCmdProcessor EXTENDS Module
VAR_INPUT
	Acceleration: LREAL:=1000.0;
	AccFactor: LREAL:=0.5;
	Jerk: LREAL:=1000.0;
	JerkFactor: LREAL:=0.5;
	Command: STRING(GVL.COMMAND_LEN):='';
END_VAR
VAR_IN_OUT
	AxisGroup: AXIS_GROUP_REF_SM3;
END_VAR
VAR_OUTPUT
	Position: SMC_POS_REF;
END_VAR
VAR
	_SequenceSetCoordTrans: INT;
	_SequenceMoveCircularAbsolute: INT;
	_SequenceMoveCircularRelative: INT;
	_SequenceMoveDirectAbsolute: INT;
	_SequenceMoveDirectRelative: INT;
	_SequenceMoveLinearAbsolute: INT;
	_SequenceMoveLinearRelative: INT;
	
	_SMC_GroupPower: SMC_GroupPower;
	_GroupPower: BOOL;
	_MC_GroupEnable: MC_GroupEnable;
	_MC_GroupDisable: MC_GroupDisable;
	_MC_GroupReset: MC_GroupReset;
	_MC_GroupHalt: MC_GroupHalt;
	_MC_GroupReadActualPosition: MC_GroupReadActualPosition;
	_SMC_SetKinConfiguration: SMC_SetKinConfiguration;
	
	_MC_MoveCircularAbsolute: MC_MoveCircularAbsolute;
	_MC_MoveCircularRelative: MC_MoveCircularRelative;
	_MC_MoveDirectAbsolute: MC_MoveDirectAbsolute;
	_MC_MoveDirectRelative: MC_MoveDirectRelative;
	_MC_MoveLinearAbsolute: MC_MoveLinearAbsolute;
	_MC_MoveLinearRelative: MC_MoveLinearRelative;
	
	_UnitModeCurrentState: PACK_ML.State;
	_MoveCommandParser: ParseMoveCmd;
	_PosRef: SMC_POS_REF;
	_PosRef2: SMC_POS_REF;
	
    // coordinate transforms
	_MC_SetCoordinateTransform: MC_SetCoordinateTransform;
	_SMC_GroupSetTool: SMC_GroupSetTool;
	_MC_COORD_REF: MC_COORD_REF;
END_VAR
VAR CONSTANT
	_STEP_DONE: 				INT := 1000;
	_STEP_IDLE: 				INT := 0000;
	_STEP_COMMAND: 				INT := 0020;
	_STEP_GROUP_POWER_ON: 		INT := 0022;
	_STEP_WAIT_POWER_ON: 		INT := 0024;
	_STEP_GROUP_ENABLE: 		INT := 0030;
	_STEP_WAIT_ENABLE: 			INT := 0035;
	_STEP_READ_POSITION: 		INT := 0040;
	_STEP_WAIT_POSITION: 		INT := 0050;
	_STEP_SET_KINEMATICS: 		INT := 0060;
	_STEP_WAIT_KINEMATICS: 		INT := 0070;
	_STEP_SET_COORD_TRANS:		INT := 0071;
	_STEP_WAIT_COORD_TRANS:		INT := 0072;
	_STEP_MOVE_TYPE:			INT := 0080;
	_STEP_WAIT_MOVE: 			INT := 0090;
	_STEP_GROUP_DISABLE: 		INT := 0100;
	_STEP_WAIT_DISABLE: 		INT := 0110;
	_STEP_GROUP_POWER_OFF: 		INT := 0120;
	_STEP_ERR: 					INT := 9999;
END_VAR

                    SUPER^();

// PackML state machine implementation
_UnitModeCurrentState := SUPER^._UnitMode.CurrentState;

//
CASE SUPER^._SeqMain OF
	
	_STEP_DONE:
		SUPER^._SeqMain := _STEP_IDLE;
		
	_STEP_IDLE:
		// wait here until commanded to start
		
	_STEP_COMMAND: // parse command
		_MoveCommandParser(Command:=Command);
		SUPER^._SeqMain := _STEP_GROUP_POWER_ON;
		
	_STEP_GROUP_POWER_ON:
		_GroupPower := TRUE;
		SUPER^._SeqMain := _STEP_WAIT_POWER_ON;
		
	_STEP_WAIT_POWER_ON:
		IF _SMC_GroupPower.Error THEN
			SUPER^.M_Error(Description:=CONCAT('Move Command Error: ',
										CONCAT(TO_STRING(_SMC_GroupPower.ErrorID),
										CONCAT(' ', SMC_ErrorString(_SMC_GroupPower.ErrorID,
													SMC_Language_Type.english)))));
			SUPER^._SeqMain := _STEP_ERR; // error step so we dont spam errors
													
		ELSIF _SMC_GroupPower.Status THEN
			SUPER^._SeqMain := _STEP_GROUP_ENABLE;
			
		END_IF
		
	_STEP_GROUP_ENABLE:
		_MC_GroupEnable.Execute := TRUE;
		SUPER^._SeqMain := _STEP_WAIT_ENABLE;
		
	_STEP_WAIT_ENABLE:
		IF NOT _MC_GroupEnable.Busy THEN // this is a hack. we need to figure out is the group is already enabled first
			SUPER^._SeqMain := _STEP_READ_POSITION;
		END_IF;
		
	_STEP_READ_POSITION: // read group position
		_PosRef.c := _MoveCommandParser.stCommand.CoordRef;
		_PosRef2.c := _MoveCommandParser.stCommand.CoordRef2;
		_MC_GroupReadActualPosition.Enable := TRUE;
		SUPER^._SeqMain := _STEP_WAIT_POSITION;
		
	_STEP_WAIT_POSITION: // wait for group read position
		IF _MC_GroupReadActualPosition.Error THEN
			SUPER^.M_Error(Description:=CONCAT('Move Command Error: ',
										CONCAT(TO_STRING(_MC_GroupReadActualPosition.ErrorID),
										CONCAT(' ', SMC_ErrorString(_MC_GroupReadActualPosition.ErrorID,
													SMC_Language_Type.english)))));
			SUPER^._SeqMain := _STEP_ERR; // error step so we dont spam errors
													
		ELSIF  _MC_GroupReadActualPosition.Valid THEN
			_MC_GroupReadActualPosition.Enable := FALSE;
			SUPER^._SeqMain := _STEP_SET_KINEMATICS;
			
		END_IF
		
	_STEP_SET_KINEMATICS: // set kinematics
		_SMC_SetKinConfiguration.Execute := TRUE;
		SUPER^._SeqMain := _STEP_WAIT_KINEMATICS;
		
	_STEP_WAIT_KINEMATICS: // wait for set kinematics
		IF _SMC_SetKinConfiguration.Error THEN
			SUPER^.M_Error(Description:=CONCAT('Move Command Error: ',
										CONCAT(TO_STRING(_SMC_SetKinConfiguration.ErrorID),
										CONCAT(' ', SMC_ErrorString(_SMC_SetKinConfiguration.ErrorID,
													SMC_Language_Type.english)))));
			SUPER^._SeqMain := _STEP_ERR; // error step so we dont spam errors
													
		ELSIF _SMC_SetKinConfiguration.Done THEN
			_SMC_SetKinConfiguration.Execute := FALSE;
			SUPER^._SeqMain := _STEP_SET_COORD_TRANS;
			
		END_IF
		
	_STEP_SET_COORD_TRANS:
		_SequenceSetCoordTrans := 1;
		SUPER^._SeqMain := _STEP_WAIT_COORD_TRANS;
	
	_STEP_WAIT_COORD_TRANS:
		IF _SequenceSetCoordTrans <= 0 THEN
			SUPER^._SeqMain := _STEP_MOVE_TYPE;
		END_IF
		
	_STEP_MOVE_TYPE: // parse move type
		IF _MoveCommandParser.stCommand.MoveType = DUT_Command_MoveType.CircularMove THEN
			IF _MoveCommandParser.stCommand.PositionType = DUT_Command_PositionType.AbsolutePosition THEN
				_SequenceMoveCircularAbsolute := 1;
			ELSIF _MoveCommandParser.stCommand.PositionType = DUT_Command_PositionType.RelativePosition THEN
				_SequenceMoveCircularRelative := 1;
			END_IF
			
		ELSIF _MoveCommandParser.stCommand.MoveType = DUT_Command_MoveType.DirectMove THEN
			IF _MoveCommandParser.stCommand.PositionType = DUT_Command_PositionType.AbsolutePosition THEN
				_SequenceMoveDirectAbsolute := 1;
			ELSIF _MoveCommandParser.stCommand.PositionType = DUT_Command_PositionType.RelativePosition THEN
				_SequenceMoveDirectRelative := 1;
			END_IF
			
		ELSIF _MoveCommandParser.stCommand.MoveType = DUT_Command_MoveType.LinearMove THEN
			IF _MoveCommandParser.stCommand.PositionType = DUT_Command_PositionType.AbsolutePosition THEN
				_SequenceMoveLinearAbsolute := 1;
			ELSIF _MoveCommandParser.stCommand.PositionType = DUT_Command_PositionType.RelativePosition THEN
				_SequenceMoveLinearRelative := 1;
			END_IF
		END_IF
		
		SUPER^._SeqMain := _STEP_WAIT_MOVE;
		
	_STEP_WAIT_MOVE: // wait for move complete
		IF _SequenceMoveCircularAbsolute = 0
			AND _SequenceMoveCircularRelative = 0 
			AND _SequenceMoveDirectAbsolute = 0 
			AND _SequenceMoveDirectRelative = 0
			AND _SequenceMoveLinearAbsolute = 0
			AND _SequenceMoveLinearRelative = 0 THEN
				SUPER^._SeqMain := _STEP_GROUP_DISABLE;
		END_IF
		
	_STEP_GROUP_DISABLE:
		_MC_GroupDisable.Execute := TRUE;
		SUPER^._SeqMain := _STEP_WAIT_DISABLE;
		
	_STEP_WAIT_DISABLE:
		IF NOT _MC_GroupDisable.Busy THEN // this is a hack. we need to figure out if the group is already disabled first
			_MC_GroupDisable.Execute := FALSE;
			SUPER^._SeqMain := _STEP_GROUP_POWER_OFF;
		END_IF
		
	_STEP_GROUP_POWER_OFF:
		_GroupPower := FALSE;
		SUPER^._SeqMain := _STEP_DONE;
	
END_CASE

CASE _SequenceMoveCircularAbsolute OF
	0: //
	
	1: //
		_MC_MoveCircularAbsolute.Execute := TRUE;
		_SequenceMoveCircularAbsolute := 2;
		
	2: //
		IF _MC_MoveCircularAbsolute.Error THEN
			SUPER^.M_Error(Description:=CONCAT('Move Command Error: ',
										CONCAT(TO_STRING(_MC_MoveCircularAbsolute.ErrorID),
										CONCAT(' ', SMC_ErrorString(_MC_MoveCircularAbsolute.ErrorID,
													SMC_Language_Type.english)))));
			_SequenceMoveCircularAbsolute := 3; // error step so we dont spam errors
		ELSIF  _MC_MoveCircularAbsolute.Done THEN
			_MC_MoveCircularAbsolute.Execute := FALSE;
			_SequenceMoveCircularAbsolute := 0;
		END_IF
		
END_CASE

CASE _SequenceMoveCircularRelative OF
	0: //
	
	1: //
		_MC_MoveCircularRelative.Execute := TRUE;
		_SequenceMoveCircularRelative := 2;
		
	2: //
		IF _MC_MoveCircularRelative.Error THEN
			SUPER^.M_Error(Description:=CONCAT('Move Command Error: ',
										CONCAT(TO_STRING(_MC_MoveCircularRelative.ErrorID),
										CONCAT(' ', SMC_ErrorString(_MC_MoveCircularRelative.ErrorID,
													SMC_Language_Type.english)))));
			_SequenceMoveCircularRelative := 3; // error step so we dont spam errors
		ELSIF  _MC_MoveCircularRelative.Done THEN
			_MC_MoveCircularRelative.Execute := FALSE;
			_SequenceMoveCircularRelative := 0;
		END_IF
		
END_CASE

CASE _SequenceMoveDirectAbsolute OF
	0: //
	
	1: //
		_MC_MoveDirectAbsolute.Execute := TRUE;
		_SequenceMoveDirectAbsolute := 2;
		
	2: //
		IF _MC_MoveDirectAbsolute.Error THEN
			SUPER^.M_Error(Description:=CONCAT('Move Command Error: ',
										CONCAT(TO_STRING(_MC_MoveDirectAbsolute.ErrorID),
										CONCAT(' ', SMC_ErrorString(_MC_MoveDirectAbsolute.ErrorID,
													SMC_Language_Type.english)))));
			_SequenceMoveDirectAbsolute := 3; // error step so we dont spam errors
			
		ELSIF _MC_MoveDirectAbsolute.Done THEN
			_MC_MoveDirectAbsolute.Execute := FALSE;
			_SequenceMoveDirectAbsolute := 0;
		END_IF
		
END_CASE

CASE _SequenceMoveDirectRelative OF
	0: //
	
	1: //
		_MC_MoveDirectRelative.Execute := TRUE;
		_SequenceMoveDirectRelative := 2;
		
	2: //
		IF _MC_MoveDirectRelative.Error THEN
			SUPER^.M_Error(Description:=CONCAT('Move Command Error: ',
										CONCAT(TO_STRING(_MC_MoveDirectRelative.ErrorID),
										CONCAT(' ', SMC_ErrorString(_MC_MoveDirectRelative.ErrorID,
													SMC_Language_Type.english)))));
			_SequenceMoveDirectRelative := 3; // error step so we dont spam errors
			
		ELSIF _MC_MoveDirectRelative.Done THEN
			_MC_MoveDirectRelative.Execute := FALSE;
			_SequenceMoveDirectRelative := 0;
		END_IF
		
END_CASE

CASE _SequenceMoveLinearAbsolute OF
	0: //
	
	1: //
		_MC_MoveLinearAbsolute.Execute := TRUE;
		_SequenceMoveLinearAbsolute := 2;
		
	2: //
		IF _MC_MoveLinearAbsolute.Error THEN
			SUPER^.M_Error(Description:=CONCAT('Move Command Error: ',
										CONCAT(TO_STRING(_MC_MoveLinearAbsolute.ErrorID),
										CONCAT(' ', SMC_ErrorString(_MC_MoveLinearAbsolute.ErrorID,
													SMC_Language_Type.english)))));
			_SequenceMoveLinearAbsolute := 3; // error step so we dont spam errors
			
		ELSIF _MC_MoveLinearAbsolute.Done THEN
			_MC_MoveLinearAbsolute.Execute := FALSE;
			_SequenceMoveLinearAbsolute := 0;
		END_IF
END_CASE

CASE _SequenceMoveLinearRelative OF
	0: //
	
	1: //
		_MC_MoveLinearRelative.Execute := TRUE;
		_SequenceMoveLinearRelative := 2;
		
	2: //
		IF _MC_MoveLinearRelative.Error THEN
		SUPER^.M_Error(Description:=CONCAT('Move Command Error: ',
										CONCAT(TO_STRING(_MC_MoveLinearRelative.ErrorID),
										CONCAT(' ', SMC_ErrorString(_MC_MoveLinearRelative.ErrorID,
													SMC_Language_Type.english)))));
			_SequenceMoveLinearRelative := 3; // error step so we dont spam errors
			
		ELSIF _MC_MoveLinearRelative.Done THEN
			_MC_MoveLinearRelative.Execute := FALSE;
			_SequenceMoveLinearRelative := 0;
		END_IF
		
END_CASE

CASE _SequenceSetCoordTrans OF
	0: //
	
	1: //
		_MC_COORD_REF := SUPER^.StoredPositions[GVL.MCS_POS_IDX].Position; // MCS
		_MC_SetCoordinateTransform.CoordSystem := SMC_COORD_SYSTEM.MCS;
		_MC_SetCoordinateTransform.Execute := TRUE;
		_SequenceSetCoordTrans := _SequenceSetCoordTrans + 1;
		
	2: //
		IF _MC_SetCoordinateTransform.Error THEN
			SUPER^.M_Error(Description:=CONCAT('Move Command Error: ',
										CONCAT(TO_STRING(_MC_SetCoordinateTransform.ErrorID),
										CONCAT(' ', SMC_ErrorString(_MC_SetCoordinateTransform.ErrorID,
													SMC_Language_Type.english)))));
			_SequenceSetCoordTrans := 10; // error step so we dont spam errors
			
		ELSIF _MC_SetCoordinateTransform.Done THEN
			_MC_SetCoordinateTransform.Execute := FALSE;
			_SequenceSetCoordTrans := _SequenceSetCoordTrans + 1;
		END_IF
		
	3: //
		_MC_COORD_REF := SUPER^.StoredPositions[GVL.PC1_POS_IDX].Position; // PCS 1
		_MC_SetCoordinateTransform.CoordSystem := SMC_COORD_SYSTEM.PCS_1;
		_MC_SetCoordinateTransform.Execute := TRUE;
		_SequenceSetCoordTrans := _SequenceSetCoordTrans + 1;
		
	4: //
		IF _MC_SetCoordinateTransform.Error THEN
			SUPER^.M_Error(Description:=CONCAT('Move Command Error: ',
										CONCAT(TO_STRING(_MC_SetCoordinateTransform.ErrorID),
										CONCAT(' ', SMC_ErrorString(_MC_SetCoordinateTransform.ErrorID,
													SMC_Language_Type.english)))));
			_SequenceSetCoordTrans := 10; // error step so we dont spam errors
			
		ELSIF _MC_SetCoordinateTransform.Done THEN
			_MC_SetCoordinateTransform.Execute := FALSE;
			_SequenceSetCoordTrans := _SequenceSetCoordTrans + 1;
		END_IF
		
	5: //
		_MC_COORD_REF := SUPER^.StoredPositions[GVL.PC2_POS_IDX].Position; // PCS 2
		_MC_SetCoordinateTransform.CoordSystem := SMC_COORD_SYSTEM.PCS_2;
		_MC_SetCoordinateTransform.Execute := TRUE;
		_SequenceSetCoordTrans := _SequenceSetCoordTrans + 1;
		
	6: //
		IF _MC_SetCoordinateTransform.Error THEN
			SUPER^.M_Error(Description:=CONCAT('Move Command Error: ',
										CONCAT(TO_STRING(_MC_SetCoordinateTransform.ErrorID),
										CONCAT(' ', SMC_ErrorString(_MC_SetCoordinateTransform.ErrorID,
													SMC_Language_Type.english)))));
			_SequenceSetCoordTrans := 10; // error step so we dont spam errors
			
		ELSIF _MC_SetCoordinateTransform.Done THEN
			_MC_SetCoordinateTransform.Execute := FALSE;
			_SequenceSetCoordTrans := _SequenceSetCoordTrans + 1;
		END_IF
		
	7:  // set tool offset
		_MC_COORD_REF := SUPER^.StoredPositions[GVL.TCP_POS_IDX].Position; // TCP
		_SMC_GroupSetTool.Execute := TRUE;
		_SequenceSetCoordTrans := _SequenceSetCoordTrans + 1;
		
	8: // monitor tool offset
		IF _SMC_GroupSetTool.Error THEN
			SUPER^.M_Error(Description:=CONCAT('Move Command Error: ',
										CONCAT(TO_STRING(_SMC_GroupSetTool.ErrorID),
										CONCAT(' ', SMC_ErrorString(_SMC_GroupSetTool.ErrorID,
													SMC_Language_Type.english)))));
			_SequenceSetCoordTrans := 10; // error step so we dont spam errors
			
		ELSIF _SMC_GroupSetTool.Done THEN
			_SMC_GroupSetTool.Execute := FALSE;
			_SequenceSetCoordTrans := 0;
		END_IF

END_CASE

_SMC_GroupPower(
	AxisGroup:= AxisGroup, 
	Enable:= _GroupPower, 
	bRegulatorOn:= _GroupPower, 
	bDriveStart:= _GroupPower, 
	Status=> , 
	Busy=> , 
	Error=> , 
	ErrorID=> );

_MC_GroupHalt(
	AxisGroup:= AxisGroup, 
	Execute:= , 
	Deceleration:= Acceleration, 
	Jerk:= Jerk, 
	AccFactor:= AccFactor, 
	JerkFactor:= JerkFactor, 
	TorqueFactor:= , 
	ClearMovements:= , 
	Done=> , 
	Busy=> , 
	Active=> , 
	CommandAborted=> , 
	CommandAccepted=> , 
	Error=> , 
	ErrorID=> , 
	MovementId=> );
_MC_GroupEnable(
	AxisGroup:= AxisGroup, 
	Execute:= , 
	CompatibilityOptions:= , 
	Done=> , 
	Busy=> , 
	Error=> , 
	ErrorID=> );
//_MC_GroupEnable.Execute := FALSE;
_MC_GroupDisable(
	AxisGroup:= AxisGroup, 
	Execute:= , 
	Done=> , 
	Busy=> , 
	Error=> , 
	ErrorID=> );
//_MC_GroupDisable.Execute := FALSE;
_MC_GroupReset(
	AxisGroup:= AxisGroup, 
	Execute:= , 
	Done=> , 
	Busy=> , 
	Error=> , 
	ErrorID=> );
//_MC_GroupReset.Execute := FALSE; this causes it to be busy on each scan
_MC_GroupReadActualPosition(
	AxisGroup:= AxisGroup, 
	Enable:= , 
	CoordSystem:= _MoveCommandParser.stCommand.CoordSystem, 
	Valid=> , 
	Busy=> , 
	Error=> , 
	ErrorID=> , 
	Position=> Position, 
	KinematicConfig=> );
	
_SMC_SetKinConfiguration(
	AxisGroup:= AxisGroup, 
	Execute:= , 
	ConfigData:= _MC_GroupReadActualPosition.KinematicConfig, 
	Done=> , 
	Busy=> , 
	Error=> , 
	ErrorID=> );

_MC_SetCoordinateTransform(
	AxisGroup:= AxisGroup, 
	Execute:= , 
	CoordTransform:= _MC_COORD_REF, 
	CoordSystem:= , 
	Done=> , 
	Busy=> , 
	Error=> , 
	ErrorID=> );

_SMC_GroupSetTool(
	AxisGroup:= AxisGroup, 
	Execute:= , 
	ToolOffset:= _MC_COORD_REF, 
	Done=> , 
	Error=> , 
	ErrorID=> );

// https://content.helpme-codesys.com/de/libs/SM3_Robotics/Current/SM3_Robotics/POUs/Movement/MC_MoveCircularAbsolute.html
// https://content.helpme-codesys.com/de/libs/SM3_Robotics/Current/SM3_Robotics/Basic-types/SMC_CIRC_MODE.html#smc-circ-mode
_MC_MoveCircularAbsolute(
	AxisGroup:= AxisGroup, 
	Execute:= , 
	CircMode:= _MoveCommandParser.stCommand.CircleMode, 
	AuxPoint:= _PosRef, 
	EndPoint:= _PosRef2, 
	PathChoice:= _MoveCommandParser.stCommand.PathChoice, 
	Velocity:= _MoveCommandParser.stCommand.Speed, 
	Acceleration:= Acceleration, 
	Deceleration:= Acceleration, 
	Jerk:= Jerk, 
	CoordSystem:= _MoveCommandParser.stCommand.CoordSystem, 
	BufferMode:= , 
	TransitionMode:= , 
	TransitionParameter:= , 
	OrientationMode:= , 
	VelFactor:= _MoveCommandParser.stCommand.Speed / 100.0,  
	AccFactor:= AccFactor, 
	JerkFactor:= JerkFactor, 
	TorqueFactor:= 1, 
	Done=> , 
	Busy=> , 
	Active=> , 
	CommandAborted=> , 
	CommandAccepted=> , 
	Error=> , 
	ErrorID=> , 
	MovementId=> );

// https://content.helpme-codesys.com/en/libs/SM3_Robotics/Current/SM3_Robotics/POUs/Movement/MC_MoveCircularRelative.html
// https://content.helpme-codesys.com/de/libs/SM3_Robotics/Current/SM3_Robotics/Basic-types/SMC_CIRC_MODE.html#smc-circ-mode
_MC_MoveCircularRelative(
	AxisGroup:= AxisGroup, 
	Execute:= , 
	CircMode:= _MoveCommandParser.stCommand.CircleMode, 
	AuxPoint:= _PosRef, 
	EndPoint:= _PosRef2, 
	PathChoice:= _MoveCommandParser.stCommand.PathChoice, 
	Velocity:= _MoveCommandParser.stCommand.Speed, 
	Acceleration:= Acceleration, 
	Deceleration:= Acceleration, 
	Jerk:= Jerk, 
	CoordSystem:= _MoveCommandParser.stCommand.CoordSystem, 
	BufferMode:= , 
	TransitionMode:= , 
	TransitionParameter:= , 
	OrientationMode:= , 
	VelFactor:= _MoveCommandParser.stCommand.Speed / 100.0,  
	AccFactor:= AccFactor, 
	JerkFactor:= JerkFactor, 
	TorqueFactor:= 1, 
	Done=> , 
	Busy=> , 
	Active=> , 
	CommandAborted=> , 
	CommandAccepted=> , 
	Error=> , 
	ErrorID=> , 
	MovementId=> );

_MC_MoveDirectAbsolute(
	AxisGroup:=AxisGroup,
	Execute:= ,
	Position:= _PosRef,
	MovementType:= ,
	CoordSystem:= _MoveCommandParser.stCommand.CoordSystem,
	BufferMode:= ,
	TransitionMode:= ,
	TransitionParameter:= ,
	VelFactor:= _MoveCommandParser.stCommand.Speed / 100.0, 
	AccFactor:= AccFactor, 
	JerkFactor:= JerkFactor, 
	TorqueFactor:= 1,
	Done=> ,
	Busy=> ,
	Active=> ,
	CommandAborted=> ,
	CommandAccepted=> ,
	Error=> ,
	ErrorID=> ,
	MovementId=> );
						
_MC_MoveDirectRelative(
	AxisGroup:= AxisGroup, 
	Execute:= , 
	Distance:= _PosRef, 
	MovementType:= , 
	CoordSystem:= _MoveCommandParser.stCommand.CoordSystem, 
	BufferMode:= , 
	TransitionMode:= , 
	TransitionParameter:= , 
	VelFactor:= _MoveCommandParser.stCommand.Speed / 100.0,  
	AccFactor:= AccFactor, 
	JerkFactor:= JerkFactor, 
	TorqueFactor:= 1, 
	Done=> , 
	Busy=> , 
	Active=> , 
	CommandAborted=> , 
	CommandAccepted=> , 
	Error=> , 
	ErrorID=> , 
	MovementId=> );
	
_MC_MoveLinearAbsolute(
	AxisGroup:= AxisGroup, 
	Execute:= , 
	Position:= _PosRef,
	Velocity:= _MoveCommandParser.stCommand.Speed, 
	Acceleration:= Acceleration, 
	Deceleration:= Acceleration, 
	Jerk:= Jerk, 
	CoordSystem:= _MoveCommandParser.stCommand.CoordSystem, 
	BufferMode:= , 
	TransitionMode:= , 
	TransitionParameter:= , 
	OrientationMode:= , 
	VelFactor:= _MoveCommandParser.stCommand.Speed / 100.0, 
	AccFactor:= AccFactor, 
	JerkFactor:= JerkFactor, 
	TorqueFactor:= 1, 
	Done=> , 
	Busy=> , 
	Active=> , 
	CommandAborted=> , 
	CommandAccepted=> , 
	Error=> , 
	ErrorID=> , 
	MovementId=> );
	
_MC_MoveLinearRelative(
	AxisGroup:= AxisGroup, 
	Execute:= , 
	Distance:= _PosRef, 
	Velocity:= _MoveCommandParser.stCommand.Speed, 
	Acceleration:= Acceleration, 
	Deceleration:= Acceleration, 
	Jerk:= Jerk, 
	CoordSystem:= _MoveCommandParser.stCommand.CoordSystem, 
	BufferMode:= , 
	TransitionMode:= , 
	TransitionParameter:= , 
	OrientationMode:= , 
	VelFactor:= _MoveCommandParser.stCommand.Speed / 100.0,  
	AccFactor:= AccFactor, 
	JerkFactor:= JerkFactor, 
	TorqueFactor:= 1, 
	Done=> , 
	Busy=> , 
	Active=> , 
	CommandAborted=> , 
	CommandAccepted=> , 
	Error=> , 
	ErrorID=> , 
	MovementId=> );
                  

METHOD PROTECTED M_Starting : BOOL
                          // here we want to clear things and get ready for the execute state
// I can consider this the "INIT" state
SUPER^._SeqMain := _STEP_COMMAND;
SUPER^.M_StateComplete();
                        
END_METHOD

METHOD PROTECTED M_Resetting : BOOL
                          CASE SUPER^._SeqResetting OF
	0:
		_MC_GroupReset.Execute := TRUE;
		_SeqResetting := _SeqResetting + 1;
	1:
		IF NOT _MC_GroupReset.Busy THEN
			_MC_GroupReset.Execute := FALSE;
			SUPER^.M_StateComplete();
			_SeqResetting := 0;
		END_IF
END_CASE
                        
END_METHOD

METHOD PROTECTED M_Idle : BOOL
                          // in this state, we want to reset all the function blocks and hang out
_GroupPower := FALSE;
_MC_GroupEnable.Execute := FALSE;
_MC_GroupDisable.Execute := FALSE;
_MC_GroupReset.Execute := FALSE;
_MC_GroupReadActualPosition.Enable := FALSE;
_SMC_SetKinConfiguration.Execute := FALSE;
_MC_SetCoordinateTransform.Execute := FALSE;
_SMC_GroupSetTool.Execute := FALSE;
_MC_MoveCircularAbsolute.Execute := FALSE;
_MC_MoveCircularRelative.Execute := FALSE;
_MC_MoveDirectAbsolute.Execute := FALSE;
_MC_MoveDirectRelative.Execute := FALSE;
_MC_MoveLinearAbsolute.Execute := FALSE;
_MC_MoveLinearRelative.Execute := FALSE;
_SequenceMoveCircularAbsolute := 0;
_SequenceMoveCircularRelative := 0;
_SequenceMoveDirectAbsolute := 0;
_SequenceMoveDirectRelative := 0;
_SequenceMoveLinearAbsolute := 0;
_SequenceMoveLinearRelative := 0;
_SequenceSetCoordTrans := 0;
SUPER^._SeqMain := 0;
                        
END_METHOD

METHOD PROTECTED M_Holding : BOOL
                          CASE SUPER^._SeqHolding OF
	0:
		_MC_MoveCircularAbsolute.Execute := FALSE;
		_MC_MoveCircularRelative.Execute := FALSE;
		_MC_MoveDirectAbsolute.Execute := FALSE;
		_MC_MoveDirectRelative.Execute := FALSE;
		_MC_MoveLinearAbsolute.Execute := FALSE;
		_MC_MoveLinearRelative.Execute := FALSE;
		_MC_GroupHalt.Execute:=TRUE;
		_SeqHolding := _SeqHolding + 1;
	1:
		IF _MC_GroupHalt.Done THEN
			_MC_GroupHalt.Execute := FALSE;
			SUPER^.M_StateComplete();
			_SeqHolding := 0;
		END_IF
		
END_CASE


                        
END_METHOD

METHOD PROTECTED M_Execute : BOOL
                          // here we want to execute our commands/jobs/etc and set completed when done.
IF SUPER^._SeqMain =_STEP_IDLE THEN
	SUPER^.M_StateComplete();
END_IF
                        
END_METHOD

METHOD PROTECTED M_Aborting : BOOL
                          CASE _SeqAborting OF
	0:
		_GroupPower := FALSE;
		_MC_GroupDisable.Execute := TRUE;
		_SeqAborting := _SeqAborting + 1;
	1:
		IF NOT _SMC_GroupPower.Busy AND NOT _MC_GroupDisable.Busy THEN
			_MC_GroupDisable.Execute := FALSE;
			SUPER^.M_StateComplete();
			_SeqAborting := 0;
		END_IF
		
END_CASE

                        
END_METHOD

METHOD PROTECTED M_Complete : BOOL
                          // once complete, reset to get back to idle
SUPER^._UnitMode.Reset();
                        
END_METHOD

METHOD PROTECTED M_Unholding : BOOL
                          // here the operator called unhold (most likely from M_Start)
_MC_GroupHalt.Execute := FALSE;
CASE _MoveCommandParser.stCommand.MoveType OF 
	DUT_Command_MoveType.DirectMove:
		IF _MoveCommandParser.stCommand.PositionType = DUT_Command_Positiontype.AbsolutePosition THEN
			_MC_MoveDirectAbsolute.Execute := TRUE;
		ELSE
			_MC_MoveDirectRelative.Execute := TRUE;
		END_IF
	DUT_Command_MoveType.LinearMove:
		IF _MoveCommandParser.stCommand.PositionType = DUT_Command_Positiontype.AbsolutePosition THEN
			_MC_MoveLinearAbsolute.Execute := TRUE;
		ELSE
			_MC_MoveLinearRelative.Execute := TRUE;
		END_IF
	DUT_Command_MoveType.CircularMove:
		IF _MoveCommandParser.stCommand.PositionType = DUT_Command_Positiontype.AbsolutePosition THEN
			_MC_MoveCircularAbsolute.Execute := TRUE;
		ELSE
			_MC_MoveCircularRelative.Execute := TRUE;
		END_IF
END_CASE
//
SUPER^.M_StateComplete();
                        
END_METHOD

METHOD PROTECTED M_SetPackML : BOOL
                          SUPER^._UnitMode(	sName := 'Move Processor',
				eInitialState := PACK_ML.State.Idle,
				xActive := TRUE);
                        
END_METHOD

METHOD PROTECTED M_Clearing : BOOL
                          _GroupPower := FALSE;
_MC_GroupEnable.Execute := FALSE;
_MC_GroupDisable.Execute := FALSE;
_MC_GroupReset.Execute := FALSE;
_MC_GroupReadActualPosition.Enable := FALSE;
_SMC_SetKinConfiguration.Execute := FALSE;
_MC_SetCoordinateTransform.Execute := FALSE;
_SMC_GroupSetTool.Execute := FALSE;
_MC_MoveCircularAbsolute.Execute := FALSE;
_MC_MoveCircularRelative.Execute := FALSE;
_MC_MoveDirectAbsolute.Execute := FALSE;
_MC_MoveDirectRelative.Execute := FALSE;
_MC_MoveLinearAbsolute.Execute := FALSE;
_MC_MoveLinearRelative.Execute := FALSE;
_SequenceMoveCircularAbsolute := 0;
_SequenceMoveCircularRelative := 0;
_SequenceMoveDirectAbsolute := 0;
_SequenceMoveDirectRelative := 0;
_SequenceMoveLinearAbsolute := 0;
_SequenceMoveLinearRelative := 0;
_SequenceSetCoordTrans := 0;

SUPER^.M_StateComplete();
                        
END_METHOD
END_FUNCTION_BLOCK

FUNCTION_BLOCK VarSetCmdProcessor EXTENDS Module
VAR_INPUT
	Command: STRING(GVL.COMMAND_LEN):='';
END_VAR
VAR_OUTPUT
END_VAR
VAR
END_VAR
VAR CONSTANT
	_STEP_DONE: 		INT := 1000;
	_STEP_IDLE: 		INT := 0000;
	_STEP_COMMAND: 		INT := 0010;
	_STEP_ERR: 			INT := 0020;
END_VAR
VAR
	_UnitModeCurrentState: PACK_ML.State;
	_VarSetCmdParser: ParseVarSetCmd;
END_VAR

                    SUPER^();

// PackML state machine implementation
_UnitModeCurrentState := SUPER^._UnitMode.CurrentState;

//
CASE SUPER^._SeqMain OF
    _STEP_DONE:
		SUPER^._SeqMain := _STEP_IDLE;
        
    _STEP_IDLE:
		// hang out here until called to run
		
	_STEP_COMMAND:
        _VarSetCmdParser(Command:=Command);
		IF _VarSetCmdParser.Error THEN
			//
			SUPER^.M_Error(Description:=_VarSetCmdParser.ErrorDescription);
			// next, please
			SUPER^._SeqMain := _STEP_ERR;
			
		ELSE
			//
			IF _VarSetCmdParser.stCommand.ArrayType = DUT_Command_ArrayType.StoredPosition THEN
				SUPER^.StoredPositions[_VarSetCmdParser.stCommand.ArrayIndex].Position := _VarSetCmdParser.stCommand.Coordinates;
			ELSIF _VarSetCmdParser.stCommand.ArrayType = DUT_Command_ArrayType.VisionRegister THEN
				SUPER^.VisionRegisters[_VarSetCmdParser.stCommand.ArrayIndex].Position := _VarSetCmdParser.stCommand.Coordinates;
			ELSIF _VarSetCmdParser.stCommand.ArrayType = DUT_Command_ArrayType.Flag THEN
				// will just let the flag take on the value of X
				SUPER^.Flags[_VarSetCmdParser.stCommand.ArrayIndex].Value := LREAL_TO_BOOL(_VarSetCmdParser.stCommand.Coordinates.X);
			END_IF
			// next, please
			SUPER^._SeqMain := _STEP_DONE;
			
		END_IF

END_CASE
                  

METHOD PROTECTED M_SetPackML : BOOL
                          SUPER^._UnitMode(	sName := 'VarSet Processor', 
				eInitialState := PACK_ML.State.Idle,
				xActive := TRUE);
                        
END_METHOD

METHOD PROTECTED M_Complete : BOOL
                          // once complete, reset to get back to idle
SUPER^._UnitMode.Reset();
                        
END_METHOD

METHOD PROTECTED M_Starting : BOOL
                          // here we want to clear things and get ready for the execute state
// I can consider this the "INIT" state
SUPER^._SeqMain := _STEP_COMMAND;
SUPER^.M_StateComplete();
                        
END_METHOD

METHOD PROTECTED M_Execute : BOOL
                          // here we want to execute our commands/jobs/etc and set completed when done.
IF SUPER^._SeqMain =_STEP_IDLE THEN
	SUPER^.M_StateComplete();
END_IF
                        
END_METHOD
END_FUNCTION_BLOCK

FUNCTION_BLOCK PauseCmdProcessor EXTENDS Module
VAR_INPUT
	Command: STRING(GVL.COMMAND_LEN):='';
END_VAR
VAR_OUTPUT
	ElapsedTime: TIME;
	RemainingTime: TIME;
END_VAR
VAR
	_Timer: TON;
	_Timer_IN: BOOL;
	_Timer_PT: TIME;
	_Timer_Q: BOOL;
	_Timer_ET: TIME;
END_VAR
VAR
	_UnitModeCurrentState: PACK_ML.State;
	_ParsePauseCmd: ParsePauseCmd;
END_VAR
VAR CONSTANT
	_STEP_DONE: 		INT := 1000;
	_STEP_IDLE: 		INT := 0000;
	_STEP_COMMAND: 		INT := 0010;
	_STEP_TWO: 			INT := 0020;
	_STEP_ERR: 			INT := 0030;
END_VAR

                    SUPER^();

// PackML state machine implementation
_UnitModeCurrentState := SUPER^._UnitMode.CurrentState;

//
CASE SUPER^._SeqMain OF
	
    _STEP_DONE:
 		_Timer_IN := FALSE;
		SUPER^._SeqMain := _STEP_IDLE;
        
    _STEP_IDLE:
		// hang out here until called to run
        
    _STEP_COMMAND:
		_ParsePauseCmd(Command:=Command);
		_Timer_PT := _ParsePauseCmd.stCommand.PauseTime;
 		_Timer_IN := TRUE;
		// next, please
		SUPER^._SeqMain := _STEP_TWO;
		
	_STEP_TWO:
		IF _Timer.Q THEN
			// next, please
			SUPER^._SeqMain := _STEP_DONE;
		END_IF

END_CASE

_Timer(
	IN:= _Timer_IN, 
	PT:= _Timer_PT, 
	Q=> _Timer_Q, 
	ET=> _Timer_ET);
	
ElapsedTime := _Timer_ET;
RemainingTime := _Timer_PT - _Timer_ET;
                  

METHOD PROTECTED M_SetPackML : BOOL
                          SUPER^._UnitMode(	sName := 'Pause Processor',
				eInitialState := PACK_ML.State.Idle,
				xActive := TRUE);
                        
END_METHOD

METHOD PROTECTED M_Complete : BOOL
                          // once complete, reset to get back to idle
SUPER^._UnitMode.Reset();
                        
END_METHOD

METHOD PROTECTED M_Resetting : BOOL
                          CASE SUPER^._SeqResetting OF
	0:
		_Timer_IN := FALSE;
		_SeqResetting := _SeqResetting + 1;
	1:
		IF NOT _Timer_IN THEN
			SUPER^.M_StateComplete();
			_SeqResetting := 0;
		END_IF
END_CASE
                        
END_METHOD

METHOD PROTECTED M_Execute : BOOL
                          // here we want to execute our commands/jobs/etc and set completed when done.
IF SUPER^._SeqMain =_STEP_IDLE THEN
	SUPER^.M_StateComplete();
END_IF
                        
END_METHOD

METHOD PROTECTED M_Starting : BOOL
                          // here we want to clear things and get ready for the execute state
// I can consider this the "INIT" state
SUPER^._SeqMain := _STEP_COMMAND;
SUPER^.M_StateComplete();
                        
END_METHOD
END_FUNCTION_BLOCK

FUNCTION_BLOCK OutputCmdProcessor EXTENDS Module
VAR_INPUT
	Enable: BOOL;
	Command: STRING(GVL.COMMAND_LEN):='';
END_VAR
VAR_IN_OUT
	Servo1: AXIS_REF_SM3;
	Servo2: AXIS_REF_SM3;
	Outputs: ARRAY [GVL.DIG_OUT_ARR_BEG..GVL.DIG_OUT_ARR_END] OF BOOL;
END_VAR
VAR_OUTPUT
END_VAR
VAR
	// servo 1
	_Servo1_Execute: BOOL;
	_Servo1_Speed: LREAL := 360;
	_Servo1_Position: LREAL := 0;
	_Servo1_MC_Power: MC_Power;
	_Servo1_MC_Halt: MC_Halt;
	_Servo1_MC_MoveAbsolute: MC_MoveAbsolute;
	
	// servo 2
	_Servo2_Execute: BOOL;
	_Servo2_Speed: LREAL := 360;
	_Servo2_Position: LREAL := 0;
	_Servo2_MC_Power: MC_Power;
	_Servo2_MC_Halt: MC_Halt;
	_Servo2_MC_MoveAbsolute: MC_MoveAbsolute;
END_VAR
VAR
	_RunRtrig: R_TRIG;
	_SequenceDigital: INT;
	_SequenceAnalog: INT;
	_SequenceServo: INT;
	
	_UnitModeCurrentState: PACK_ML.State;
	_OutputCommandParser: ParseOutputCmd;
	_OutputType: DUT_OutputType;
	_OutputTarget: INT;
	_OutputValue1, _OutputValue2: LREAL;
END_VAR
VAR CONSTANT
	_STEP_DONE: 		INT := 1000;
	_STEP_IDLE: 		INT := 0000;
	_STEP_COMMAND: 		INT := 0010;
	_STEP_TWO: 			INT := 0020;
	_STEP_ERR: 			INT := 0030;
END_VAR

                    SUPER^();

// PackML state machine implementation
_UnitModeCurrentState := SUPER^._UnitMode.CurrentState;

//
CASE SUPER^._SeqMain OF
	
    _STEP_DONE:
		SUPER^._SeqMain := _STEP_IDLE;
        
    _STEP_IDLE:
        // hang out here untill called to run
		
    _STEP_COMMAND:
		_OutputCommandParser(Command:=Command);
		IF _OutputCommandParser.Error THEN
			SUPER^.M_Error(Description:=_OutputCommandParser.ErrorDescription);
			SUPER^._SeqMain := _STEP_ERR;
		ELSE
			_OutputType := _OutputCommandParser.stCommand.OutputType;
			_OutputTarget := _OutputCommandParser.stCommand.OutputTarget;
			_OutputValue1 := _OutputCommandParser.stCommand.OutputValue1;
			_OutputValue2 := _OutputCommandParser.stCommand.OutputValue2;
			
			CASE _OutputType OF
				DUT_OutputType.Digital: //
					_SequenceDigital := 1;
					SUPER^._SeqMain := _STEP_TWO;
				DUT_OutputType.Analog: //
					_SequenceAnalog := 1;
					SUPER^._SeqMain := _STEP_TWO;
				DUT_OutputType.Servo: //
					_SequenceServo := 1;
					SUPER^._SeqMain := _STEP_TWO;
			ELSE
				SUPER^._SeqMain := _STEP_DONE;
				
			END_CASE
		END_IF
		
	_STEP_TWO:
		IF _SequenceDigital = 0 
			AND _SequenceAnalog = 0
			AND _SequenceServo = 0 THEN
				// next, please
				SUPER^._SeqMain := _STEP_DONE;
		END_IF;

END_CASE

CASE _SequenceDigital OF
	0: //
	1: //
		THIS^.Outputs[_OutputTarget] := _OutputValue1 > 0;
		_SequenceDigital := 0;
END_CASE

CASE _SequenceAnalog OF
	0: //
	1: //
		CASE _OutputTarget OF
			0: //
				// set analog value here
				// i got nothing right now
				_SequenceAnalog := 0;
		END_CASE
	2: //
END_CASE

CASE _SequenceServo OF
	0: //
	1: //
		CASE _OutputTarget OF
			0: //
				_SequenceServo := 0;
			1: //
				_Servo1_Execute := TRUE;
				_Servo1_Position := _OutputValue1;
				_Servo1_Speed := _OutputValue2;
				_SequenceServo := 2;
			2: //
				_Servo2_Execute := TRUE;
				_Servo2_Position := _OutputValue1;
				_Servo2_Speed := _OutputValue2;
				_SequenceServo := 2;
		END_CASE
	2: //
		IF (_Servo1_Execute AND _Servo1_MC_MoveAbsolute.Done)
			OR (_Servo2_Execute AND _Servo2_MC_MoveAbsolute.Done) THEN
			_SequenceServo := 0;
			
		ELSIF _Servo1_MC_Power.Error THEN
			SUPER^.M_Error(Description:=CONCAT('Output Servo Command Error: ',
											CONCAT(TO_STRING(_Servo1_MC_Power.ErrorID),
											CONCAT(' ', SMC_ErrorString(_Servo1_MC_Power.ErrorID,
														SMC_Language_Type.english)))));
			_SequenceServo := 3;
														
		ELSIF _Servo1_MC_MoveAbsolute.Error THEN
			SUPER^.M_Error(Description:=CONCAT('Output Servo Command Error: ',
											CONCAT(TO_STRING(_Servo1_MC_MoveAbsolute.ErrorID),
											CONCAT(' ', SMC_ErrorString(_Servo1_MC_MoveAbsolute.ErrorID,
														SMC_Language_Type.english)))));
			_SequenceServo := 3;
														
		ELSIF _Servo2_MC_Power.Error THEN
			SUPER^.M_Error(Description:=CONCAT('Output Servo Command Error: ',
											CONCAT(TO_STRING(_Servo2_MC_Power.ErrorID),
											CONCAT(' ', SMC_ErrorString(_Servo2_MC_Power.ErrorID,
														SMC_Language_Type.english)))));
			_SequenceServo := 3;
														
		ELSIF _Servo1_MC_MoveAbsolute.Error THEN
			SUPER^.M_Error(Description:=CONCAT('Output Servo Command Error: ',
											CONCAT(TO_STRING(_Servo1_MC_MoveAbsolute.ErrorID),
											CONCAT(' ', SMC_ErrorString(_Servo1_MC_MoveAbsolute.ErrorID,
														SMC_Language_Type.english)))));
			_SequenceServo := 3;
		END_IF
END_CASE

// servo 1
_Servo1_MC_Power(
	Axis:= Servo1, 
	Enable:= Enable, 
	bRegulatorOn:= Enable, 
	bDriveStart:= Enable, 
	Status=> , 
	bRegulatorRealState=> , 
	bDriveStartRealState=> , 
	Busy=> , 
	Error=> , 
	ErrorID=> );
	
_Servo1_MC_MoveAbsolute(
	Axis:= Servo1, 
	Execute:= _Servo1_Execute, 
	Position:= _Servo1_Position, 
	Velocity:= _Servo1_Speed, 
	Acceleration:= 1000, 
	Deceleration:= 1000, 
	Jerk:= 1000, 
	Direction:= , 
	BufferMode:= , 
	Done=> , 
	Busy=> , 
	Active=> , 
	CommandAborted=> , 
	Error=> , 
	ErrorID=> );
	
_Servo1_MC_Halt(
	Axis:= Servo1, 
	Execute:= , 
	Deceleration:= 1000, 
	Jerk:= 1000, 
	Done=> , 
	Busy=> , 
	CommandAborted=> , 
	Error=> , 
	ErrorID=> );

// servo 2
_Servo2_MC_Power(
	Axis:= Servo2, 
	Enable:= Enable, 
	bRegulatorOn:= Enable, 
	bDriveStart:= Enable, 
	Status=> , 
	bRegulatorRealState=> , 
	bDriveStartRealState=> , 
	Busy=> , 
	Error=> , 
	ErrorID=> );
	
_Servo2_MC_MoveAbsolute(
	Axis:= Servo2, 
	Execute:= _Servo2_Execute, 
	Position:= _Servo2_Position, 
	Velocity:= _Servo2_Speed, 
	Acceleration:= 1000, 
	Deceleration:= 1000, 
	Jerk:= 1000, 
	Direction:= , 
	BufferMode:= , 
	Done=> , 
	Busy=> , 
	Active=> , 
	CommandAborted=> , 
	Error=> , 
	ErrorID=> );
	
_Servo2_MC_Halt(
	Axis:= Servo2, 
	Execute:= , 
	Deceleration:= 1000, 
	Jerk:= 1000, 
	Done=> , 
	Busy=> , 
	CommandAborted=> , 
	Error=> , 
	ErrorID=> );
                  

METHOD PROTECTED M_SetPackML : BOOL
                          SUPER^._UnitMode(	sName := 'Output Processor',
				eInitialState := PACK_ML.State.Idle,
				xActive := TRUE);
                        
END_METHOD

METHOD PROTECTED M_Resetting : BOOL
                          CASE SUPER^._SeqResetting OF
	0:
		_Servo1_Execute := FALSE;
		_Servo2_Execute := FALSE;
		_SeqResetting := _SeqResetting + 1;
	1:
		IF NOT _Servo1_MC_MoveAbsolute.Busy 
			AND NOT _Servo2_MC_MoveAbsolute.Busy  THEN
				SUPER^.M_StateComplete();
				_SeqResetting := 0;
		END_IF
END_CASE
                        
END_METHOD

METHOD PROTECTED M_Execute : BOOL
                          // here we want to execute our commands/jobs/etc and set completed when done.
IF SUPER^._SeqMain =_STEP_IDLE THEN
	SUPER^.M_StateComplete();
END_IF
                        
END_METHOD

METHOD PROTECTED M_Starting : BOOL
                          // here we want to clear things and get ready for the execute state
// I can consider this the "INIT" state
SUPER^._SeqMain := _STEP_COMMAND;
SUPER^.M_StateComplete();
                        
END_METHOD

METHOD PROTECTED M_Holding : BOOL
                          CASE SUPER^._SeqHolding OF
	0:
		_Servo1_Execute := FALSE;
		_Servo2_Execute := FALSE;
		_Servo1_MC_Halt.Execute := TRUE;
		_Servo2_MC_Halt.Execute := TRUE;
		SUPER^._SeqHolding := SUPER^._SeqHolding + 1;
	1:
		IF _Servo1_MC_Halt.Done AND _Servo2_MC_Halt.Done THEN
			_Servo1_MC_Halt.Execute := FALSE;
			_Servo2_MC_Halt.Execute := FALSE;
			SUPER^.M_StateComplete();
			SUPER^._SeqHolding := 0;
		END_IF
		
END_CASE
                        
END_METHOD

METHOD PROTECTED M_Idle : BOOL
                          _Servo1_Execute := FALSE;
_Servo2_Execute := FALSE;
_Servo1_MC_Halt.Execute := FALSE;
_Servo2_MC_Halt.Execute := FALSE;
_SequenceDigital := 0;
_SequenceAnalog := 0;
_SequenceServo := 0;
SUPER^._SeqMain := 0;
                        
END_METHOD

METHOD PROTECTED M_Unholding : BOOL
                          //
_Servo1_MC_Halt.Execute := FALSE;
_Servo2_MC_Halt.Execute := FALSE;

//
SUPER^._SeqMain := _STEP_COMMAND;

//
SUPER^.M_StateComplete();
                        
END_METHOD

METHOD PROTECTED M_Aborting : BOOL
                          CASE SUPER^._SeqAborting OF
	0:
		_Servo1_Execute := FALSE;
		_Servo2_Execute := FALSE;
		SUPER^._SeqAborting := SUPER^._SeqAborting + 1;
	1:
		IF NOT _Servo1_MC_MoveAbsolute.Busy 
			AND NOT _Servo2_MC_MoveAbsolute.Busy  THEN
				SUPER^.M_StateComplete();
				SUPER^._SeqAborting := 0;
		END_IF
		
END_CASE

                        
END_METHOD

METHOD PROTECTED M_Clearing : BOOL
                          _Servo1_Execute := FALSE;
_Servo2_Execute := FALSE;
_Servo1_MC_Halt.Execute := FALSE;
_Servo2_MC_Halt.Execute := FALSE;
_SequenceDigital := 0;
_SequenceAnalog := 0;
_SequenceServo := 0;

SUPER^.M_StateComplete();
                        
END_METHOD

METHOD PROTECTED M_Complete : BOOL
                          // once complete, reset to get back to idle
SUPER^._UnitMode.Reset();
                        
END_METHOD
END_FUNCTION_BLOCK

FUNCTION_BLOCK PackML
VAR_INPUT
END_VAR
VAR_OUTPUT
	IUnitMode: PACK_ML.IUnitMode;
END_VAR
VAR
	_UnitMode: PACK_ML.UnitMode;
	_StateTimer: TON;
	_PackMLFirstScan: BOOL:=TRUE;
	_SeqMain, _SeqAborting, _SeqClearing, _SeqCompleting, _SeqHolding, _SeqResetting,
	_SeqStarting, _SeqStopping, _SeqSuspending, _SeqUnholding, _SeqUnSuspending: INT;
END_VAR
VAR CONSTANT
	STATE_TIME: TIME := T#0MS;
END_VAR

                    //
IF _PackMLFirstScan THEN
	_PackMLFirstScan := FALSE;
	M_SetPackMl();
	IUnitMode := _UnitMode;
END_IF

//
_StateTimer(PT:=STATE_TIME);

//
CASE _UnitMode.CurrentState OF
	PACK_ML.State.Stopped:
		M_Stopped();
	PACK_ML.State.Aborted:
		M_Aborted();
	PACK_ML.State.Held:
		M_Held();
	PACK_ML.State.Suspended:
		M_Suspended();
	PACK_ML.State.Complete:
		M_Complete();
	PACK_ML.State.Idle:
		M_Idle();
	PACK_ML.State.Resetting:
		M_Resetting();
	PACK_ML.State.Starting:
		M_Starting();
	PACK_ML.State.Execute:
		M_Execute();
	PACK_ML.State.Suspending:
		M_Suspending();
	PACK_ML.State.UnSuspending:
		M_UnSuspending();
	PACK_ML.State.Holding:
		M_Holding();
	PACK_ML.State.UnHolding:
		M_UnHolding();
	PACK_ML.State.Completing:
		M_Completing();
	PACK_ML.State.Aborting:
		M_Aborting();
	PACK_ML.State.Stopping:
		M_Stopping();
	PACK_ML.State.Clearing:
		M_Clearing();
END_CASE
                  

METHOD PROTECTED M_Aborting : BOOL
VAR_INPUT
END_VAR
                          _StateTimer.IN:=TRUE;

IF _StateTimer.Q THEN
	_StateTimer.IN:=FALSE;
	M_StateComplete();
END_IF
                        
END_METHOD

METHOD PROTECTED M_Unholding : BOOL
VAR_INPUT
END_VAR
                          _StateTimer.IN:=TRUE;

IF _StateTimer.Q THEN
	_StateTimer.IN:=FALSE;
	M_StateComplete();
END_IF
                        
END_METHOD

METHOD PROTECTED M_Aborted : BOOL
VAR_INPUT
END_VAR
                          _SeqMain := 0;
_SeqAborting := 0;
_SeqClearing := 0;
_SeqCompleting := 0;
_SeqHolding := 0;
_SeqResetting := 0;
_SeqStarting := 0;
_SeqStopping := 0;
_SeqSuspending := 0;
_SeqUnholding := 0;
_SeqUnSuspending := 0;
                        
END_METHOD

METHOD PROTECTED M_Held : BOOL
VAR_INPUT
END_VAR
                          (*_StateTimer.IN:=TRUE;

IF _StateTimer.Q THEN
	_StateTimer.IN:=FALSE;
	M_StateComplete();
END_IF*)
                        
END_METHOD

METHOD PROTECTED M_Completing : BOOL
VAR_INPUT
END_VAR
                          _StateTimer.IN:=TRUE;

IF _StateTimer.Q THEN
	_StateTimer.IN:=FALSE;
	M_StateComplete();
END_IF
                        
END_METHOD

METHOD PROTECTED M_Stopping : BOOL
VAR_INPUT
END_VAR
                          _StateTimer.IN:=TRUE;

IF _StateTimer.Q THEN
	_StateTimer.IN:=FALSE;
	M_StateComplete();
END_IF
                        
END_METHOD

METHOD PROTECTED M_Clearing : BOOL
VAR_INPUT
END_VAR
                          _StateTimer.IN:=TRUE;

IF _StateTimer.Q THEN
	_StateTimer.IN:=FALSE;
	M_StateComplete();
END_IF
                        
END_METHOD

METHOD PROTECTED M_Stopped : BOOL
VAR_INPUT
END_VAR
                          (*_StateTimer.IN:=TRUE;

IF _StateTimer.Q THEN
	_StateTimer.IN:=FALSE;
	M_StateComplete();
END_IF*)
                        
END_METHOD

METHOD PROTECTED M_SetPackML : BOOL
VAR_INPUT
END_VAR
                          _UnitMode(sName := 'Normal Operation', 
			dwSupportedStates := PACK_ML.State.All,
			dwAllowsLeavingFromStates := PACK_ML.State.Stopped 
											OR PACK_ML.State.Aborted 
											OR PACK_ML.State.Idle, 
			dwAllowsEnteringIntoStates := PACK_ML.State.Stopped
											OR PACK_ML.State.Aborted 
											OR PACK_ML.State.Idle, 
			eInitialState := PACK_ML.State.Idle,
			xActive := TRUE);
                        
END_METHOD

METHOD PROTECTED M_Complete : BOOL
VAR_INPUT
END_VAR
                          (*_StateTimer.IN:=TRUE;

IF _StateTimer.Q THEN
	_StateTimer.IN:=FALSE;
	M_StateComplete();
END_IF*)
                        
END_METHOD

METHOD PROTECTED M_Resetting : BOOL
VAR_INPUT
END_VAR
                          _StateTimer.IN:=TRUE;

IF _StateTimer.Q THEN
	_StateTimer.IN:=FALSE;
	M_StateComplete();
END_IF
                        
END_METHOD

METHOD PROTECTED M_Suspended : BOOL
VAR_INPUT
END_VAR
                          (*_StateTimer.IN:=TRUE;

IF _StateTimer.Q THEN
	_StateTimer.IN:=FALSE;
	M_StateComplete();
END_IF*)
                        
END_METHOD

METHOD PROTECTED M_StateComplete : BOOL
VAR_INPUT
END_VAR
                          _UnitMode.ActingStateCompleted();
                        
END_METHOD

METHOD PROTECTED M_Suspending : BOOL
VAR_INPUT
END_VAR
                          _StateTimer.IN:=TRUE;

IF _StateTimer.Q THEN
	_StateTimer.IN:=FALSE;
	M_StateComplete();
END_IF
                        
END_METHOD

METHOD PROTECTED M_Idle : BOOL
VAR_INPUT
END_VAR
                          (*_StateTimer.IN:=TRUE;

IF _StateTimer.Q THEN
	_StateTimer.IN:=FALSE;
	M_StateComplete();
END_IF*)
                        
END_METHOD

METHOD PROTECTED M_Starting : BOOL
VAR_INPUT
END_VAR
                          _StateTimer.IN:=TRUE;

IF _StateTimer.Q THEN
	_StateTimer.IN:=FALSE;
	M_StateComplete();
END_IF
                        
END_METHOD

METHOD PROTECTED M_Execute : BOOL
VAR_INPUT
END_VAR
                          
                        
END_METHOD

METHOD PROTECTED M_UnSuspending : BOOL
VAR_INPUT
END_VAR
                          _StateTimer.IN:=TRUE;

IF _StateTimer.Q THEN
	_StateTimer.IN:=FALSE;
	M_StateComplete();
END_IF
                        
END_METHOD

METHOD PROTECTED M_Holding : BOOL
VAR_INPUT
END_VAR
                          _StateTimer.IN:=TRUE;

IF _StateTimer.Q THEN
	_StateTimer.IN:=FALSE;
	M_StateComplete();
END_IF
                        
END_METHOD
END_FUNCTION_BLOCK

FUNCTION_BLOCK CncCmdProcessor EXTENDS Module
VAR_INPUT
	GapVelocity: LREAL := 10;
	AvoidGaps: BOOL := TRUE;
	GapAccel: LREAL := 500.0;
	Command: STRING(GVL.COMMAND_LEN):='';
END_VAR
VAR_IN_OUT
	AxisGroup: AXIS_GROUP_REF_SM3;
	SM3_Drive_PosControl_J1: SM3_Drive_PosControl.AXIS_REF_POSCONTROL;
	SM3_Drive_PosControl_J2: SM3_Drive_PosControl.AXIS_REF_POSCONTROL;
	SM3_Drive_PosControl_J3: SM3_Drive_PosControl.AXIS_REF_POSCONTROL;
	SM3_Drive_PosControl_J4: SM3_Drive_PosControl.AXIS_REF_POSCONTROL;
	SM3_Drive_PosControl_J5: SM3_Drive_PosControl.AXIS_REF_POSCONTROL;
	SM3_Drive_PosControl_J6: SM3_Drive_PosControl.AXIS_REF_POSCONTROL;
END_VAR
VAR_OUTPUT
END_VAR
VAR
	_SMC_TrafoConfig_ArticulatedRobot_6DOF: SMC_TrafoConfig_ArticulatedRobot_6DOF;
	_SMC_Trafo_ArticulatedRobot_6DOF: SMC_Trafo_ArticulatedRobot_6DOF;
	_SMC_Trafof_ArticulatedRobot_6DOF: SMC_Trafof_ArticulatedRobot_6DOF;
	_SMC_ControlAxisByPos_J1: SMC_ControlAxisByPos;
	_SMC_ControlAxisByPos_J2: SMC_ControlAxisByPos;
	_SMC_ControlAxisByPos_J3: SMC_ControlAxisByPos;
	_SMC_ControlAxisByPos_J4: SMC_ControlAxisByPos;
	_SMC_ControlAxisByPos_J5: SMC_ControlAxisByPos;
	_SMC_ControlAxisByPos_J6: SMC_ControlAxisByPos;
	_SMC_Interpolator: SMC_Interpolator;
	_PlanPath: CncPathPlanner;
	_ErrorRtrig: R_TRIG;
END_VAR
VAR CONSTANT
	wVarCount : WORD := 1;
END_VAR
VAR
	lrR1 : LREAL:=30;
	
	astVar : ARRAY [0..wVarCount] OF SMC_SingleVar :=
			[(strVarName:='R1', pAdr := ADR(lrR1), eVarType := SMC_VarType.SMC_TYPE_LREAL)];
			
	stVarList : SMC_VarList := (wNumberVars := wVarCount, psvVarlist := ADR(astVar));
END_VAR
VAR CONSTANT
	_STEP_DONE: 		INT := 1000;
	_STEP_IDLE: 		INT := 0000;
	_STEP_COMMAND: 		INT := 0010;
	_STEP_ONE: 			INT := 0020;
END_VAR
VAR
	_UnitModeCurrentState: PACK_ML.State;
	_CncCmdParser: ParseCncCmd;
END_VAR

                    // NOTE currently the settings for J6 invert direction under scaling/mapping contradict using motion control 
// libraries and CNC. For CNC to work properly, the setting is required to be enabled (inverted). Additionally
// the homing direction and position will need to be negated. This all requires a full download. Will be leaving 
// setting disabled for now so that we can continue to use motion control. 
//
// to recap, take these steps if you would like to try out CNC:
// 1. open the axis pool settings and under the scaling/mapping section enable 'invert direction'
// 2. in the A_Homing POU, change the homing direction to positive.
// 3. in _00_MAIN POU, under FirstScan set the initial home offset to a positive value (keep the value and just change the sign).
// 4. do a full download.
// 5. go online and set the persistent value (if previously initialized in FirstScan) to a positive value.
//
// UPDATE: Figured out a work around for this issue. In the A_Interpolater POU, I negated the set position in the ControlAxisByPos
// function block for J6 such that it drives the opposite way. This appears to have resolved the issue. Why this is needed, I do not
// know. I am sure it is some minor overlooked detail somewhere in the code...

SUPER^();

// PackML state machine implementation
_UnitModeCurrentState := SUPER^._UnitMode.CurrentState;

//
CASE SUPER^._SeqMain OF
    _STEP_DONE:
		_SMC_Interpolator.bExecute := FALSE;
		SUPER^._SeqMain := _STEP_IDLE;
        
    _STEP_IDLE:
		// hang out here until called to start
	
	_STEP_COMMAND:
		//
		_CncCmdParser(Command:=Command);	
		_PlanPath.M_SetOriConvention(OriConvention:=_CncCmdParser.stCommand.OriConvention);
		_PlanPath.M_SetStartPosition(StartPos:=_CncCmdParser.stCommand.StartPos);
		_PlanPath.M_Execute(Filename:=_CncCmdParser.stCommand.Filename); // TODO I think we should be careful here. May need to sync CheckVelocities with the Interpolator
		
		//
		IF NOT _CncCmdParser.Error THEN
			_SMC_Interpolator.bExecute := TRUE;
			SUPER^._SeqMain := _STEP_ONE;
		ELSE
			SUPER^.M_Error(Description:=CONCAT('Command parsing error: ',_CncCmdParser.ErrorDescription));
		END_IF
        
    _STEP_ONE:
		IF NOT _SMC_Interpolator.bBusy AND NOT SUPER^.Error THEN
			// next, please
			SUPER^._SeqMain := _STEP_DONE;
		END_IF

END_CASE

// TODO these should reference INOUT AxisGroup but somehow wont compile like that. 
// using global scoped vars for now
_SMC_TrafoConfig_ArticulatedRobot_6DOF.a1:=ArfBotAxisGroup.Trafo.a1;//AxisGroup.Trafo.a1;
_SMC_TrafoConfig_ArticulatedRobot_6DOF.a2:=ArfBotAxisGroup.Trafo.a2;//AxisGroup.Trafo.a2;
_SMC_TrafoConfig_ArticulatedRobot_6DOF.a3:=ArfBotAxisGroup.Trafo.a3;//AxisGroup.Trafo.a3;
// conflicting documentation on if d1 needs to be pos or neg. only works as negative otherwise trafo reports invalid configuration
// https://product-help.schneider-electric.com/Machine%20Expert/V2.0/zh/codesys_softmotion/codesys_softmotion/modules/_sm_trafo_pou_six_dof_robot.html
// https://forge.codesys.com/forge/talk/Motion/thread/16e1f0327f/
_SMC_TrafoConfig_ArticulatedRobot_6DOF.d1:=-ArfBotAxisGroup.Trafo.d1;//-AxisGroup.Trafo.d1;
_SMC_TrafoConfig_ArticulatedRobot_6DOF.d3:=ArfBotAxisGroup.Trafo.d3;//AxisGroup.Trafo.d3;
_SMC_TrafoConfig_ArticulatedRobot_6DOF.d4:=ArfBotAxisGroup.Trafo.d4;//AxisGroup.Trafo.d4;
_SMC_TrafoConfig_ArticulatedRobot_6DOF.d6:=ArfBotAxisGroup.Trafo.d6;//AxisGroup.Trafo.d6;
_SMC_TrafoConfig_ArticulatedRobot_6DOF.q3_max_deg:=160; // TODO put magic numbers somewhere appropriate
_SMC_TrafoConfig_ArticulatedRobot_6DOF.q3_min_deg:=-160; // TODO put magic numbers somewhere appropriate
_SMC_TrafoConfig_ArticulatedRobot_6DOF.q5_max_deg:=160; // TODO put magic numbers somewhere appropriate
_SMC_TrafoConfig_ArticulatedRobot_6DOF.q5_min_deg:=-160; // TODO put magic numbers somewhere appropriate


// TODO figure out how this var list can be used. for now its just hello world
_PlanPath(VarList:= stVarList, DataOut=> );

_SMC_Interpolator.bEmergency_Stop := _SMC_ControlAxisByPos_J1.bError OR _SMC_ControlAxisByPos_J1.bStopIpo
									OR _SMC_ControlAxisByPos_J2.bError OR _SMC_ControlAxisByPos_J2.bStopIpo
									OR _SMC_ControlAxisByPos_J3.bError OR _SMC_ControlAxisByPos_J3.bStopIpo
									OR _SMC_ControlAxisByPos_J4.bError OR _SMC_ControlAxisByPos_J4.bStopIpo
									OR _SMC_ControlAxisByPos_J5.bError OR _SMC_ControlAxisByPos_J5.bStopIpo
									OR _SMC_ControlAxisByPos_J6.bError OR _SMC_ControlAxisByPos_J6.bStopIpo;

_SMC_Interpolator(
	bExecute:= , 
	poqDataIn:= _PlanPath.DataOut, 
	bSlow_Stop:= , 
	bEmergency_Stop:= , 
	bWaitAtNextStop:= , 
	dOverride:= , 
	iVelMode:= , 
	dwIpoTime:= GVL.dwMainInterval, // in microseconds and should match the task time
	dLastWayPos:= , 
	bAbort:= NOT _SMC_Interpolator.bExecute, 
	bSingleStep:= , 
	bAcknM:= , 
	bQuick_Stop:= , 
	dQuickDeceleration:= , 
	dJerkMax:= , 
	dQuickStopJerk:= , 
	bSuppressSystemMFunctions:= , 
	bDone=> , 
	bBusy=> , 
	bError=> , 
	wErrorID=> , 
	piSetPosition=> , 
	iStatus=> , 
	bWorking=> , 
	iActObjectSourceNo=> , 
	dActObjectLength=> , 
	dActObjectLengthRemaining=> , 
	dVel=> , 
	vecActTangent=> , 
	iLastSwitch=> , 
	dwSwitches=> , 
	dWayPos=> , 
	wM=> , 
	adToolLength=> , 
	Act_Object=> );

// handle m codes
CASE _SMC_Interpolator.wM OF
	0:	// rest acknowledgment
		_SMC_Interpolator.bAcknM := FALSE;
	200: // close gripper
		_SMC_Interpolator.bAcknM := TRUE;
		GVL.Servo0Position := 0; // TODO
	201: // open gripper
		_SMC_Interpolator.bAcknM := TRUE;
		GVL.Servo0Position := 255; // TODO
END_CASE

_SMC_Trafo_ArticulatedRobot_6DOF(
	config:= _SMC_TrafoConfig_ArticulatedRobot_6DOF, 
	pi:= _SMC_Interpolator.piSetPosition, 
	dQ0_old:= SM_Drive_PosControl_J1.fActPosition, 
	dQ1_old:= SM_Drive_PosControl_J2.fActPosition, 
	dQ2_old:= SM_Drive_PosControl_J3.fActPosition, 
	dQ3_old:= SM_Drive_PosControl_J4.fActPosition, 
	dQ4_old:= SM_Drive_PosControl_J5.fActPosition, 
	dQ5_old:= SM_Drive_PosControl_J6.fActPosition, 
	armState:= , 
	elbowState:= , 
	handState:= , 
	dQ0=> , 
	dQ1=> , 
	dQ2=> , 
	dQ3=> , 
	dQ4=> , 
	dQ5=> , 
	bError=> , 
	result=> );
	
_SMC_ControlAxisByPos_J1(
	Axis:= SM3_Drive_PosControl_J1, 
	iStatus:= _SMC_Interpolator.iStatus, 
	bEnable:= _SMC_Interpolator.bWorking, 
	bAvoidGaps:= AvoidGaps, 
	fSetPosition:= _SMC_Trafo_ArticulatedRobot_6DOF.dQ0, 
	fGapVelocity:= GapVelocity, 
	fGapAcceleration:= GapAccel, 
	fGapDeceleration:= GapAccel, 
	fGapJerk:= , 
	bBusy=> , 
	bCommandAborted=> , 
	bError=> , 
	iErrorID=> , 
	bStopIpo=> );
	
_SMC_ControlAxisByPos_J2(
	Axis:= SM3_Drive_PosControl_J2, 
	iStatus:= _SMC_Interpolator.iStatus, 
	bEnable:= _SMC_Interpolator.bWorking, 
	bAvoidGaps:= AvoidGaps, 
	fSetPosition:= _SMC_Trafo_ArticulatedRobot_6DOF.dQ1, 
	fGapVelocity:= GapVelocity, 
	fGapAcceleration:= GapAccel, 
	fGapDeceleration:= GapAccel, 
	fGapJerk:= , 
	bBusy=> , 
	bCommandAborted=> , 
	bError=> , 
	iErrorID=> , 
	bStopIpo=> );
	
_SMC_ControlAxisByPos_J3(
	Axis:= SM3_Drive_PosControl_J3, 
	iStatus:= _SMC_Interpolator.iStatus, 
	bEnable:= _SMC_Interpolator.bWorking, 
	bAvoidGaps:= AvoidGaps, 
	fSetPosition:= _SMC_Trafo_ArticulatedRobot_6DOF.dQ2, 
	fGapVelocity:= GapVelocity, 
	fGapAcceleration:= GapAccel, 
	fGapDeceleration:= GapAccel, 
	fGapJerk:= , 
	bBusy=> , 
	bCommandAborted=> , 
	bError=> , 
	iErrorID=> , 
	bStopIpo=> );
	
_SMC_ControlAxisByPos_J4(
	Axis:= SM3_Drive_PosControl_J4, 
	iStatus:= _SMC_Interpolator.iStatus, 
	bEnable:= _SMC_Interpolator.bWorking, 
	bAvoidGaps:= AvoidGaps, 
	fSetPosition:= _SMC_Trafo_ArticulatedRobot_6DOF.dQ3, 
	fGapVelocity:= GapVelocity, 
	fGapAcceleration:= GapAccel, 
	fGapDeceleration:= GapAccel, 
	fGapJerk:= , 
	bBusy=> , 
	bCommandAborted=> , 
	bError=> , 
	iErrorID=> , 
	bStopIpo=> );
	
_SMC_ControlAxisByPos_J5(
	Axis:= SM3_Drive_PosControl_J5, 
	iStatus:= _SMC_Interpolator.iStatus, 
	bEnable:= _SMC_Interpolator.bWorking, 
	bAvoidGaps:= AvoidGaps, 
	fSetPosition:= _SMC_Trafo_ArticulatedRobot_6DOF.dQ4, 
	fGapVelocity:= GapVelocity, 
	fGapAcceleration:= GapAccel, 
	fGapDeceleration:= GapAccel, 
	fGapJerk:= , 
	bBusy=> , 
	bCommandAborted=> , 
	bError=> , 
	iErrorID=> , 
	bStopIpo=> );
	
_SMC_ControlAxisByPos_J6(
	Axis:= SM3_Drive_PosControl_J6, 
	iStatus:= _SMC_Interpolator.iStatus, 
	bEnable:= _SMC_Interpolator.bWorking, 
	bAvoidGaps:= AvoidGaps, 
	fSetPosition:= -_SMC_Trafo_ArticulatedRobot_6DOF.dQ5, // please see note in A_CNC POU regarding why this was set to negative
	fGapVelocity:= GapVelocity, 
	fGapAcceleration:= GapAccel, 
	fGapDeceleration:= GapAccel, 
	fGapJerk:= , 
	bBusy=> , 
	bCommandAborted=> , 
	bError=> , 
	iErrorID=> , 
	bStopIpo=> );
	
_ErrorRtrig();
_ErrorRtrig.CLK := _PlanPath.Error
					OR _SMC_Interpolator.bError
					OR _SMC_Trafo_ArticulatedRobot_6DOF.bError
					OR _SMC_ControlAxisByPos_J1.bError
					OR _SMC_ControlAxisByPos_J2.bError
					OR _SMC_ControlAxisByPos_J3.bError
					OR _SMC_ControlAxisByPos_J4.bError
					OR _SMC_ControlAxisByPos_J5.bError
					OR _SMC_ControlAxisByPos_J6.bError;
IF _ErrorRtrig.Q THEN
	IF _PlanPath.Error THEN
		SUPER^.M_Error(Description:=_PlanPath.ErrorDescription);
	END_IF
	IF _SMC_Interpolator.bError THEN
		SUPER^.M_Error(Description := CONCAT(' Interpolator Error: ',
                                CONCAT(TO_STRING(_SMC_Interpolator.wErrorID),
                                CONCAT(' ', SMC_ErrorString(_SMC_Interpolator.wErrorID,
                                            SMC_Language_Type.english)))));
	END_IF
	IF _SMC_Trafo_ArticulatedRobot_6DOF.bError THEN
		SUPER^.M_Error(Description := CONCAT(' Trafo Error: ', 'unknown'));
	END_IF
	IF _SMC_ControlAxisByPos_J1.bError THEN
		SUPER^.M_Error(Description := CONCAT(' ControlAxisByPos_J1 Error: ',
                                CONCAT(TO_STRING(_SMC_ControlAxisByPos_J1.iErrorID),
                                CONCAT(' ', SMC_ErrorString(_SMC_ControlAxisByPos_J1.iErrorID,
                                            SMC_Language_Type.english)))));
	END_IF
	IF _SMC_ControlAxisByPos_J2.bError THEN
		SUPER^.M_Error(Description := CONCAT(' ControlAxisByPos_J2 Error: ',
                                CONCAT(TO_STRING(_SMC_ControlAxisByPos_J2.iErrorID),
                                CONCAT(' ', SMC_ErrorString(_SMC_ControlAxisByPos_J2.iErrorID,
                                            SMC_Language_Type.english)))));
	END_IF
	IF _SMC_ControlAxisByPos_J3.bError THEN
		SUPER^.M_Error(Description := CONCAT(' ControlAxisByPos_J3 Error: ',
                                CONCAT(TO_STRING(_SMC_ControlAxisByPos_J3.iErrorID),
                                CONCAT(' ', SMC_ErrorString(_SMC_ControlAxisByPos_J3.iErrorID,
                                            SMC_Language_Type.english)))));
	END_IF
	IF _SMC_ControlAxisByPos_J4.bError THEN
		SUPER^.M_Error(Description := CONCAT(' ControlAxisByPos_J4 Error: ',
                                CONCAT(TO_STRING(_SMC_ControlAxisByPos_J4.iErrorID),
                                CONCAT(' ', SMC_ErrorString(_SMC_ControlAxisByPos_J4.iErrorID,
                                            SMC_Language_Type.english)))));
	END_IF
	IF _SMC_ControlAxisByPos_J5.bError THEN
		SUPER^.M_Error(Description := CONCAT(' ControlAxisByPos_J5 Error: ',
                                CONCAT(TO_STRING(_SMC_ControlAxisByPos_J5.iErrorID),
                                CONCAT(' ', SMC_ErrorString(_SMC_ControlAxisByPos_J5.iErrorID,
                                            SMC_Language_Type.english)))));
	END_IF
	IF _SMC_ControlAxisByPos_J6.bError THEN
		SUPER^.M_Error(Description := CONCAT(' ControlAxisByPos_J6 Error: ',
                                CONCAT(TO_STRING(_SMC_ControlAxisByPos_J6.iErrorID),
                                CONCAT(' ', SMC_ErrorString(_SMC_ControlAxisByPos_J6.iErrorID,
                                            SMC_Language_Type.english)))));
	END_IF
END_IF
                  

METHOD PROTECTED M_SetPackML : BOOL
                          SUPER^._UnitMode(	sName := 'CNC Processor',
				eInitialState := PACK_ML.State.Idle,
				xActive := TRUE);
                        
END_METHOD

METHOD PROTECTED M_Complete : BOOL
                          // once complete, reset to get back to idle
SUPER^._UnitMode.Reset();
                        
END_METHOD

METHOD PROTECTED M_Execute : BOOL
                          // here we want to execute our commands/jobs/etc and set completed when done.
IF SUPER^._SeqMain =_STEP_IDLE THEN
	SUPER^.M_StateComplete();
END_IF
                        
END_METHOD

METHOD PROTECTED M_Starting : BOOL
                          // here we want to clear things and get ready for the execute state
// I can consider this the "INIT" state
SUPER^._SeqMain := _STEP_COMMAND;
SUPER^.M_StateComplete();
                        
END_METHOD

METHOD PROTECTED M_Resetting : BOOL
                          CASE SUPER^._SeqResetting OF
	0:
		_PlanPath.M_Reset();
		_SeqResetting := _SeqResetting + 1;
	1:
		IF NOT _PlanPath.Error THEN
			SUPER^.M_StateComplete();
			_SeqResetting := 0;
		END_IF
END_CASE
                        
END_METHOD

METHOD PROTECTED M_Holding : BOOL
                          CASE _SeqHolding OF
	0:
		_SMC_Interpolator.bWaitAtNextStop := TRUE;
		SUPER^._SeqHolding := SUPER^._SeqHolding + 1;
	1:
		// TODO dale thomas this is not tested
		IF NOT _SMC_Interpolator.bWorking THEN
			SUPER^._SeqHolding := 0;
			SUPER^.M_StateComplete();
		END_IF
		
END_CASE


                        
END_METHOD

METHOD PROTECTED M_Unholding : BOOL
                          CASE _SeqUnHolding OF
	0:
		_SMC_Interpolator.bWaitAtNextStop := FALSE;
		SUPER^._SeqUnHolding := SUPER^._SeqUnHolding + 1;
	1:
		// TODO dale thomas this is not tested
		IF _SMC_Interpolator.bWorking THEN
			SUPER^._SeqUnHolding := 0;
			SUPER^.M_StateComplete();
		END_IF
		
END_CASE
                        
END_METHOD

METHOD PROTECTED M_Idle : BOOL
                          _SMC_Interpolator.bWaitAtNextStop := FALSE;
_SMC_Interpolator.bExecute := FALSE;
                        
END_METHOD
END_FUNCTION_BLOCK

FUNCTION_BLOCK ParseCncCmd
VAR_INPUT
	Command: STRING(GVL.COMMAND_LEN);
END_VAR
VAR_OUTPUT
	stCommand: ST_CncCmd;
	Error: BOOL:= FALSE;
	ErrorDescription: STRING;
END_VAR
VAR
	_CmdParams: ARRAY [0..GVL.COMMAND_LEN] OF STRING;
END_VAR
VAR CONSTANT
	_AddString: STRING(3):='ADD';
	_XYZString: STRING(3):='XYZ';
	_ZYXString: STRING(3):='ZYX';
	_ZYZString: STRING(3):='ZYZ';
	_LiteralString: STRING(3):='LIT';
	_VariableString: STRING(3):='VAR';
	_StoredPositionsString: STRING(3):='STO';
	_VisionRegistersString: STRING(3):='VIS';
	_FlagsString: STRING(3):='FLG';
END_VAR

                    // /path/to/file/with/no/spaces/file.cnc ADD|XYX|ZYX|ZYZ startpos
// file1.cnc XYZ H +0250.00 +0000.00 +0500.00 +0000.00 +0045.00 +0180.00
// file2.cnc ADD A S 025
// file3.cnc ADD A V 015

Error := FALSE;
ErrorDescription:='';

// split command string into commands
_CmdParams:=F_SplitCmd(Command:=Command);

//
IF _CmdParams[0] <> '' THEN
	//
	stCommand.Filename:=_CmdParams[0];
	
	//
	IF _CmdParams[1] = _AddString THEN
		stCommand.OriConvention := SMC_ORI_CONVENTION.ADDAXES;
	ELSIF _CmdParams[1] = _XYZString THEN
		stCommand.OriConvention := SMC_ORI_CONVENTION.XYZ;
	ELSIF _CmdParams[1] = _ZYXString THEN
		stCommand.OriConvention := SMC_ORI_CONVENTION.ZYX;
	ELSIF _CmdParams[1] = _ZYZString THEN
		stCommand.OriConvention := SMC_ORI_CONVENTION.ZYZ;
	ELSE
		Error := TRUE;
		ErrorDescription:='No ori convention provided';
	END_IF
	
